C07287=1050.995,70.390,419.955,170.839,33.457,156.282
C07288=1051.001,70.640,419.937,170.841,33.459,156.283
C07289=1051.007,70.890,419.919,170.843,33.461,156.283
C07290=1051.013,71.138,419.901,170.844,33.463,156.283
C07291=1051.019,71.388,419.883,170.846,33.465,156.284
C07292=1051.025,71.638,419.865,170.847,33.467,156.284
C07293=1051.031,71.887,419.846,170.849,33.469,156.284
C07294=1051.037,72.136,419.828,170.851,33.471,156.285
C07295=1051.044,72.385,419.810,170.852,33.473,156.285
C07296=1051.050,72.635,419.792,170.854,33.475,156.285
C07297=1051.056,72.884,419.775,170.856,33.478,156.286
C07298=1051.062,73.133,419.756,170.857,33.479,156.286
C07299=1051.068,73.382,419.738,170.859,33.481,156.286
C07300=1051.075,73.632,419.720,170.861,33.483,156.287
C07301=1051.080,73.881,419.702,170.863,33.485,156.287
C07302=1051.086,74.130,419.684,170.865,33.487,156.287
C07303=1051.093,74.379,419.665,170.866,33.490,156.288
C07304=1051.099,74.629,419.648,170.868,33.492,156.288
C07305=1051.105,74.878,419.629,170.870,33.494,156.288
C07306=1051.111,75.127,419.611,170.871,33.496,156.289
C07307=1051.117,75.376,419.593,170.873,33.498,156.289
C07308=1051.124,75.626,419.575,170.874,33.500,156.289
C07309=1051.130,75.874,419.557,170.876,33.502,156.290
C07310=1051.136,76.124,419.539,170.878,33.504,156.290
C07311=1051.142,76.373,419.520,170.879,33.506,156.291
C07312=1051.148,76.623,419.503,170.881,33.508,156.291
C07313=1051.154,76.871,419.484,170.883,33.510,156.291
C07314=1051.160,77.121,419.466,170.884,33.512,156.291
C07315=1051.167,77.407,419.445,170.886,33.515,156.292
C07316=1051.175,77.693,419.424,170.888,33.517,156.292
C07317=1051.182,77.978,419.403,170.890,33.519,156.293
C07318=1051.189,78.264,419.382,170.892,33.522,156.293
C07319=1051.195,78.513,419.364,170.893,33.524,156.293
C07320=1051.201,78.762,419.346,170.895,33.526,156.294
C07321=1051.207,79.011,419.327,170.897,33.528,156.294
C07322=1051.213,79.261,419.309,170.898,33.530,156.294
C07323=1051.219,79.510,419.290,170.900,33.532,156.295
C07324=1051.225,79.759,419.271,170.901,33.534,156.295
C07325=1051.231,80.009,419.254,170.903,33.536,156.295
C07326=1051.237,80.257,419.235,170.905,33.538,156.296
C07327=1051.244,80.506,419.217,170.906,33.541,156.296
C07328=1051.250,80.756,419.199,170.908,33.543,156.297
C07329=1051.255,81.006,419.179,170.909,33.545,156.297
C07330=1051.262,81.255,419.161,170.911,33.547,156.297
C07331=1051.267,81.504,419.143,170.913,33.549,156.298
C07332=1051.274,81.753,419.125,170.914,33.551,156.298
C07333=1051.280,82.002,419.106,170.916,33.553,156.298
C07334=1051.286,82.252,419.087,170.918,33.555,156.299
C07335=1051.292,82.501,419.069,170.919,33.558,156.299
C07336=1051.298,82.750,419.050,170.921,33.560,156.299
C07337=1051.304,82.999,419.032,170.922,33.562,156.300
C07338=1051.310,83.249,419.014,170.924,33.564,156.300
C07339=1051.316,83.498,418.995,170.926,33.566,156.300
C07340=1051.322,83.747,418.976,170.927,33.568,156.301
C07341=1051.329,83.996,418.957,170.929,33.570,156.301
C07342=1051.335,84.246,418.939,170.931,33.572,156.301
C07343=1051.340,84.495,418.920,170.933,33.574,156.302
C07344=1051.347,84.744,418.902,170.935,33.576,156.302
C07345=1051.353,84.993,418.883,170.936,33.579,156.302
C07346=1051.359,85.242,418.865,170.938,33.580,156.303
C07347=1051.365,85.492,418.847,170.940,33.582,156.303
C07348=1051.371,85.741,418.827,170.941,33.584,156.303
C07349=1051.378,85.990,418.809,170.943,33.586,156.304
C07350=1051.384,86.239,418.790,170.945,33.589,156.304
C07351=1051.390,86.489,418.771,170.946,33.591,156.304
C07352=1051.396,86.738,418.752,170.948,33.593,156.305
C07353=1051.402,86.987,418.735,170.949,33.595,156.305
C07354=1051.408,87.236,418.716,170.951,33.597,156.305
C07355=1051.415,87.485,418.697,170.953,33.599,156.306
C07356=1051.420,87.735,418.678,170.954,33.601,156.306
C07357=1051.427,87.984,418.659,170.956,33.603,156.307
C07358=1051.433,88.233,418.641,170.958,33.605,156.307
C07359=1051.439,88.482,418.622,170.959,33.607,156.307
C07360=1051.445,88.732,418.603,170.961,33.609,156.307
C07361=1051.452,88.981,418.584,170.963,33.612,156.308
C07362=1051.458,89.230,418.566,170.964,33.614,156.308
C07363=1051.464,89.480,418.548,170.966,33.616,156.309
C07364=1051.470,89.729,418.528,170.968,33.618,156.309
C07365=1051.476,89.978,418.510,170.969,33.620,156.309
C07366=1051.483,90.227,418.491,170.971,33.622,156.310
C07367=1051.489,90.476,418.472,170.972,33.624,156.310
C07368=1051.495,90.726,418.453,170.974,33.626,156.310
C07369=1051.501,90.975,418.435,170.976,33.628,156.311
C07370=1051.507,91.224,418.415,170.977,33.631,156.311
C07371=1051.513,91.473,418.397,170.979,33.633,156.311
C07372=1051.519,91.723,418.377,170.981,33.634,156.312
C07373=1051.525,91.972,418.359,170.982,33.636,156.312
C07374=1051.531,92.221,418.340,170.984,33.639,156.312
C07375=1051.537,92.469,418.321,170.985,33.641,156.313
C07376=1051.543,92.719,418.301,170.988,33.643,156.313
C07377=1051.549,92.968,418.283,170.990,33.645,156.314
C07378=1051.555,93.217,418.263,170.991,33.647,156.314
C07379=1051.562,93.504,418.242,170.993,33.650,156.314
C07380=1051.569,93.789,418.220,170.995,33.652,156.315
C07381=1051.576,94.075,418.198,170.997,33.655,156.315
C07382=1051.583,94.360,418.176,170.999,33.657,156.315
C07383=1051.589,94.609,418.158,171.000,33.659,156.316
C07384=1051.595,94.858,418.138,171.002,33.662,156.316
C07385=1051.602,95.107,418.119,171.004,33.664,156.317
C07386=1051.608,95.356,418.100,171.005,33.666,156.317
C07387=1051.613,95.606,418.080,171.007,33.667,156.317
C07388=1051.620,95.855,418.062,171.009,33.670,156.318
C07389=1051.625,96.104,418.043,171.010,33.672,156.318
C07390=1051.632,96.353,418.024,171.012,33.674,156.318
C07391=1051.638,96.602,418.004,171.014,33.676,156.319
C07392=1051.644,96.851,417.985,171.015,33.678,156.319
C07393=1051.650,97.101,417.966,171.017,33.680,156.319
C07394=1051.656,97.350,417.947,171.019,33.682,156.320
C07395=1051.662,97.599,417.928,171.020,33.684,156.320
C07396=1051.669,97.848,417.909,171.022,33.687,156.320
C07397=1051.674,98.097,417.890,171.024,33.689,156.321
C07398=1051.680,98.347,417.870,171.025,33.691,156.321
C07399=1051.687,98.597,417.851,171.027,33.693,156.321
C07400=1051.693,98.845,417.831,171.028,33.695,156.322
C07401=1051.700,99.094,417.813,171.030,33.697,156.322
C07402=1051.705,99.344,417.793,171.032,33.699,156.323
C07403=1051.712,99.592,417.774,171.033,33.701,156.323
C07404=1051.718,99.842,417.755,171.036,33.704,156.323
C07405=1051.724,100.091,417.736,171.038,33.706,156.324
C07406=1051.730,100.340,417.717,171.039,33.708,156.324
C07407=1051.736,100.589,417.697,171.041,33.710,156.324
C07408=1051.742,100.838,417.678,171.043,33.712,156.325
C07409=1051.748,101.088,417.659,171.044,33.714,156.325
C07410=1051.754,101.337,417.639,171.046,33.716,156.325
C07411=1051.760,101.587,417.620,171.048,33.719,156.326
C07412=1051.767,101.835,417.600,171.049,33.721,156.326
C07413=1051.773,102.085,417.581,171.051,33.723,156.326
C07414=1051.778,102.334,417.562,171.053,33.725,156.327
C07415=1051.784,102.583,417.542,171.054,33.727,156.327
C07416=1051.790,102.832,417.522,171.056,33.729,156.328
C07417=1051.797,103.081,417.503,171.058,33.732,156.328
C07418=1051.802,103.330,417.484,171.059,33.733,156.328
C07419=1051.808,103.579,417.464,171.061,33.735,156.329
C07420=1051.814,103.829,417.445,171.062,33.738,156.329
C07421=1051.821,104.078,417.424,171.064,33.740,156.329
C07422=1051.826,104.327,417.405,171.066,33.742,156.330
C07423=1051.833,104.576,417.386,171.067,33.744,156.330
C07424=1051.839,104.825,417.367,171.069,33.746,156.330
C07425=1051.845,105.074,417.347,171.071,33.748,156.331
C07426=1051.850,105.324,417.327,171.072,33.751,156.331
C07427=1051.856,105.572,417.307,171.074,33.753,156.332
C07428=1051.863,105.822,417.289,171.076,33.755,156.332
C07429=1051.869,106.071,417.268,171.078,33.757,156.332
C07430=1051.875,106.321,417.249,171.080,33.759,156.333
C07431=1051.881,106.569,417.229,171.082,33.761,156.333
C07432=1051.887,106.819,417.210,171.083,33.764,156.333
C07433=1051.893,107.068,417.190,171.085,33.766,156.334
C07434=1051.899,107.317,417.171,171.087,33.768,156.334
C07435=1051.906,107.566,417.151,171.088,33.770,156.335
C07436=1051.912,107.815,417.131,171.090,33.772,156.335
C07437=1051.918,108.064,417.112,171.092,33.774,156.335
C07438=1051.924,108.313,417.092,171.093,33.777,156.336
C07439=1051.929,108.563,417.073,171.095,33.779,156.336
C07440=1051.936,108.812,417.052,171.097,33.781,156.336
C07441=1051.943,109.061,417.033,171.098,33.783,156.337
C07442=1051.948,109.310,417.014,171.100,33.785,156.337
C07443=1051.955,109.596,416.991,171.102,33.788,156.337
C07444=1051.963,109.881,416.968,171.104,33.790,156.338
C07445=1051.970,110.166,416.946,171.106,33.792,156.338
C07446=1051.976,110.452,416.923,171.108,33.795,156.339
C07447=1051.982,110.701,416.903,171.110,33.797,156.339
C07448=1051.988,110.951,416.883,171.111,33.799,156.339
C07449=1051.994,111.200,416.863,171.113,33.801,156.340
C07450=1052.000,111.449,416.843,171.115,33.803,156.340
C07451=1052.006,111.698,416.824,171.117,33.806,156.341
C07452=1052.012,111.947,416.804,171.119,33.808,156.341
C07453=1052.019,112.197,416.784,171.121,33.810,156.341
C07454=1052.025,112.445,416.764,171.122,33.812,156.342
C07455=1052.030,112.695,416.745,171.124,33.814,156.342
C07456=1052.036,112.944,416.725,171.126,33.816,156.342
C07457=1052.043,113.193,416.704,171.127,33.819,156.343
C07458=1052.049,113.442,416.684,171.129,33.821,156.343
C07459=1052.055,113.691,416.665,171.131,33.823,156.343
C07460=1052.061,113.940,416.645,171.132,33.825,156.344
C07461=1052.067,114.190,416.625,171.134,33.827,156.344
C07462=1052.073,114.439,416.605,171.136,33.830,156.345
C07463=1052.079,114.688,416.584,171.137,33.831,156.345
C07464=1052.085,114.936,416.564,171.139,33.834,156.345
C07465=1052.091,115.186,416.544,171.141,33.836,156.346
C07466=1052.097,115.435,416.525,171.142,33.838,156.346
C07467=1052.102,115.685,416.504,171.144,33.840,156.346
C07468=1052.108,115.933,416.484,171.146,33.843,156.347
C07469=1052.115,116.183,416.464,171.147,33.845,156.347
C07470=1052.121,116.432,416.444,171.149,33.847,156.348
C07471=1052.126,116.681,416.423,171.152,33.849,156.348
C07472=1052.132,116.930,416.403,171.154,33.852,156.348
C07473=1052.139,117.179,416.383,171.155,33.854,156.349
C07474=1052.144,117.428,416.363,171.157,33.856,156.349
C07475=1052.150,117.677,416.343,171.159,33.858,156.349
C07476=1052.156,117.926,416.323,171.160,33.860,156.350
C07477=1052.162,118.175,416.302,171.162,33.863,156.350
C07478=1052.168,118.424,416.282,171.164,33.865,156.351
C07479=1052.174,118.673,416.262,171.165,33.867,156.351
C07480=1052.180,118.923,416.241,171.167,33.869,156.351
C07481=1052.186,119.172,416.221,171.169,33.872,156.352
C07482=1052.191,119.421,416.201,171.170,33.874,156.352
C07483=1052.197,119.670,416.181,171.172,33.876,156.352
C07484=1052.204,119.919,416.161,171.174,33.878,156.353
C07485=1052.210,120.168,416.141,171.176,33.880,156.353
C07486=1052.215,120.417,416.120,171.177,33.883,156.354
C07487=1052.222,120.667,416.100,171.179,33.885,156.354
C07488=1052.228,120.915,416.080,171.181,33.887,156.354
C07489=1052.233,121.165,416.059,171.182,33.889,156.355
C07490=1052.240,121.414,416.039,171.185,33.892,156.355
C07491=1052.246,121.663,416.019,171.187,33.894,156.356
C07492=1052.252,121.912,415.997,171.188,33.896,156.356
C07493=1052.258,122.161,415.977,171.190,33.898,156.356
C07494=1052.264,122.410,415.957,171.192,33.900,156.357
C07495=1052.270,122.659,415.937,171.194,33.903,156.357
C07496=1052.276,122.908,415.917,171.195,33.905,156.357
C07497=1052.282,123.157,415.897,171.197,33.907,156.358
C07498=1052.288,123.407,415.876,171.199,33.909,156.358
C07499=1052.294,123.656,415.856,171.200,33.911,156.358
C07500=1052.300,123.905,415.835,171.202,33.914,156.359
C07501=1052.306,124.153,415.815,171.204,33.916,156.359
C07502=1052.312,124.403,415.794,171.206,33.918,156.360
C07503=1052.318,124.652,415.774,171.207,33.920,156.360
C07504=1052.324,124.901,415.754,171.209,33.922,156.360
C07505=1052.330,125.150,415.732,171.211,33.925,156.361
C07506=1052.336,125.399,415.712,171.213,33.926,156.361
C07507=1052.343,125.684,415.689,171.215,33.929,156.362
C07508=1052.350,125.970,415.666,171.218,33.932,156.362
C07509=1052.357,126.256,415.642,171.220,33.934,156.362
C07510=1052.364,126.541,415.618,171.222,33.937,156.363
C07511=1052.370,126.790,415.598,171.223,33.939,156.363
C07512=1052.377,127.039,415.577,171.225,33.941,156.364
C07513=1052.382,127.288,415.557,171.227,33.943,156.364
C07514=1052.389,127.537,415.537,171.229,33.945,156.364
C07515=1052.394,127.786,415.515,171.230,33.948,156.365
C07516=1052.401,128.036,415.495,171.232,33.950,156.365
C07517=1052.407,128.284,415.475,171.234,33.952,156.366
C07518=1052.413,128.534,415.454,171.236,33.954,156.366
C07519=1052.419,128.782,415.433,171.237,33.956,156.366
C07520=1052.426,129.032,415.413,171.239,33.958,156.367
C07521=1052.431,129.281,415.392,171.241,33.960,156.367
C07522=1052.438,129.530,415.371,171.243,33.963,156.367
C07523=1052.444,129.779,415.352,171.244,33.965,156.368
C07524=1052.450,130.028,415.330,171.246,33.967,156.368
C07525=1052.456,130.277,415.310,171.249,33.969,156.369
C07526=1052.462,130.527,415.289,171.251,33.971,156.369
C07527=1052.468,130.775,415.268,171.252,33.973,156.369
C07528=1052.475,131.024,415.248,171.254,33.976,156.370
C07529=1052.481,131.273,415.226,171.256,33.978,156.370
C07530=1052.487,131.522,415.206,171.258,33.980,156.370
C07531=1052.493,131.772,415.185,171.259,33.982,156.371
C07532=1052.499,132.020,415.165,171.261,33.985,156.371
C07533=1052.505,132.270,415.144,171.263,33.987,156.371
C07534=1052.511,132.519,415.123,171.265,33.989,156.372
C07535=1052.517,132.768,415.102,171.266,33.991,156.372
C07536=1052.523,133.017,415.081,171.268,33.994,156.373
C07537=1052.529,133.266,415.060,171.270,33.996,156.373
C07538=1052.535,133.515,415.039,171.272,33.998,156.373
C07539=1052.541,133.764,415.018,171.273,34.000,156.374
C07540=1052.546,134.013,414.997,171.275,34.003,156.374
C07541=1052.553,134.262,414.976,171.278,34.005,156.375
C07542=1052.559,134.511,414.956,171.280,34.007,156.375
C07543=1052.565,134.760,414.934,171.282,34.009,156.375
C07544=1052.571,135.009,414.914,171.283,34.012,156.376
C07545=1052.577,135.258,414.892,171.285,34.014,156.376
C07546=1052.582,135.507,414.871,171.287,34.016,156.377
C07547=1052.589,135.756,414.851,171.289,34.018,156.377
C07548=1052.595,136.005,414.829,171.290,34.021,156.377
C07549=1052.600,136.255,414.809,171.292,34.022,156.378
C07550=1052.607,136.503,414.788,171.294,34.025,156.378
C07551=1052.613,136.752,414.766,171.296,34.027,156.378
C07552=1052.619,137.002,414.745,171.298,34.030,156.379
C07553=1052.625,137.250,414.725,171.299,34.031,156.379
C07554=1052.631,137.499,414.703,171.301,34.034,156.380
C07555=1052.637,137.749,414.682,171.303,34.036,156.380
C07556=1052.643,137.998,414.661,171.306,34.038,156.380
C07557=1052.650,138.246,414.640,171.307,34.041,156.381
C07558=1052.655,138.496,414.619,171.309,34.043,156.381
C07559=1052.661,138.745,414.598,171.311,34.045,156.382
C07560=1052.667,138.994,414.576,171.313,34.047,156.382
C07561=1052.673,139.242,414.555,171.315,34.050,156.382
C07562=1052.679,139.492,414.534,171.316,34.052,156.383
C07563=1052.685,139.741,414.513,171.318,34.054,156.383
C07564=1052.691,139.990,414.492,171.320,34.056,156.384
C07565=1052.697,140.239,414.470,171.322,34.059,156.384
C07566=1052.702,140.488,414.449,171.324,34.061,156.384
C07567=1052.709,140.737,414.428,171.325,34.063,156.385
C07568=1052.715,140.986,414.407,171.327,34.066,156.385
C07569=1052.721,141.235,414.385,171.329,34.068,156.386
C07570=1052.727,141.484,414.364,171.332,34.070,156.386
C07571=1052.733,141.770,414.340,171.334,34.073,156.386
C07572=1052.741,142.054,414.315,171.336,34.075,156.387
C07573=1052.747,142.339,414.290,171.338,34.078,156.387
C07574=1052.754,142.625,414.266,171.340,34.081,156.388
C07575=1052.760,142.874,414.244,171.342,34.083,156.388
C07576=1052.767,143.123,414.223,171.344,34.086,156.389
C07577=1052.772,143.372,414.202,171.345,34.088,156.389
C07578=1052.778,143.621,414.180,171.347,34.090,156.389
C07579=1052.785,143.870,414.159,171.349,34.092,156.390
C07580=1052.790,144.119,414.137,171.351,34.095,156.390
C07581=1052.796,144.368,414.116,171.353,34.097,156.391
C07582=1052.802,144.617,414.094,171.355,34.099,156.391
C07583=1052.808,144.866,414.074,171.357,34.102,156.391
C07584=1052.814,145.115,414.052,171.359,34.103,156.392
C07585=1052.820,145.365,414.030,171.361,34.106,156.392
C07586=1052.826,145.614,414.009,171.363,34.108,156.393
C07587=1052.832,145.862,413.987,171.365,34.111,156.393
C07588=1052.838,146.111,413.966,171.367,34.113,156.393
C07589=1052.844,146.361,413.944,171.368,34.115,156.394
C07590=1052.850,146.609,413.923,171.370,34.117,156.394
C07591=1052.856,146.858,413.901,171.372,34.119,156.395
C07592=1052.862,147.108,413.880,171.374,34.122,156.395
C07593=1052.868,147.357,413.858,171.376,34.124,156.395
C07594=1052.874,147.605,413.836,171.378,34.126,156.396
C07595=1052.880,147.854,413.814,171.379,34.129,156.396
C07596=1052.886,148.103,413.793,171.381,34.131,156.397
C07597=1052.892,148.352,413.771,171.384,34.133,156.397
C07598=1052.898,148.601,413.750,171.386,34.136,156.397
C07599=1052.904,148.850,413.728,171.388,34.138,156.398
C07600=1052.910,149.099,413.707,171.390,34.140,156.398
C07601=1052.917,149.348,413.685,171.391,34.143,156.399
C07602=1052.922,149.597,413.664,171.393,34.145,156.399
C07603=1052.928,149.846,413.641,171.395,34.147,156.399
C07604=1052.934,150.095,413.619,171.397,34.150,156.400
C07605=1052.940,150.344,413.597,171.399,34.152,156.400
C07606=1052.946,150.593,413.576,171.401,34.154,156.401
C07607=1052.952,150.842,413.555,171.403,34.157,156.401
C07608=1052.958,151.090,413.532,171.404,34.159,156.401
C07609=1052.964,151.340,413.510,171.407,34.161,156.402
C07610=1052.970,151.589,413.488,171.409,34.164,156.402
C07611=1052.975,151.838,413.467,171.411,34.166,156.403
C07612=1052.982,152.086,413.445,171.413,34.168,156.403
C07613=1052.988,152.336,413.423,171.415,34.171,156.404
C07614=1052.994,152.585,413.401,171.417,34.173,156.404
C07615=1053.000,152.834,413.379,171.418,34.175,156.404
C07616=1053.006,153.082,413.357,171.420,34.178,156.405
C07617=1053.012,153.331,413.336,171.422,34.180,156.405
C07618=1053.018,153.581,413.314,171.424,34.182,156.406
C07619=1053.023,153.830,413.292,171.426,34.185,156.406
C07620=1053.030,154.079,413.269,171.428,34.187,156.406
C07621=1053.036,154.328,413.248,171.431,34.189,156.407
C07622=1053.042,154.576,413.226,171.433,34.192,156.407
C07623=1053.047,154.825,413.204,171.434,34.194,156.408
C07624=1053.053,155.074,413.182,171.436,34.196,156.408
C07625=1053.060,155.323,413.160,171.438,34.199,156.409
C07626=1053.065,155.573,413.137,171.440,34.201,156.409
C07627=1053.071,155.822,413.116,171.442,34.203,156.409
C07628=1053.077,156.070,413.094,171.444,34.206,156.410
C07629=1053.083,156.319,413.071,171.446,34.208,156.410
C07630=1053.089,156.568,413.049,171.448,34.211,156.411
C07631=1053.095,156.817,413.027,171.450,34.213,156.411
C07632=1053.101,157.066,413.005,171.451,34.215,156.411
C07633=1053.107,157.315,412.983,171.454,34.218,156.412
C07634=1053.113,157.564,412.961,171.456,34.220,156.412
C07635=1053.120,157.849,412.936,171.458,34.223,156.413
C07636=1053.127,158.134,412.911,171.461,34.225,156.413
C07637=1053.134,158.418,412.885,171.463,34.228,156.414
C07638=1053.141,158.704,412.860,171.465,34.231,156.414
C07639=1053.146,158.952,412.837,171.467,34.233,156.415
C07640=1053.152,159.201,412.815,171.469,34.236,156.415
C07641=1053.158,159.450,412.792,171.471,34.238,156.415
C07642=1053.164,159.700,412.771,171.473,34.241,156.416
C07643=1053.171,159.948,412.748,171.475,34.243,156.416
C07644=1053.176,160.198,412.726,171.477,34.245,156.417
C07645=1053.183,160.446,412.704,171.479,34.248,156.417
C07646=1053.189,160.695,412.682,171.481,34.250,156.417
C07647=1053.194,160.944,412.659,171.483,34.252,156.418
C07648=1053.200,161.193,412.636,171.485,34.255,156.418
C07649=1053.206,161.443,412.614,171.487,34.257,156.419
C07650=1053.212,161.691,412.592,171.489,34.260,156.419
C07651=1053.217,161.940,412.569,171.491,34.262,156.420
C07652=1053.223,162.189,412.547,171.493,34.265,156.420
C07653=1053.228,162.438,412.524,171.495,34.267,156.421
C07654=1053.235,162.687,412.502,171.498,34.270,156.421
C07655=1053.241,162.935,412.479,171.499,34.272,156.422
C07656=1053.246,163.185,412.456,171.501,34.275,156.422
C07657=1053.252,163.434,412.434,171.503,34.277,156.422
C07658=1053.258,163.682,412.411,171.505,34.280,156.423
C07659=1053.264,163.931,412.388,171.507,34.282,156.423
C07660=1053.269,164.181,412.366,171.509,34.285,156.424
C07661=1053.274,164.429,412.343,171.511,34.287,156.424
C07662=1053.281,164.678,412.321,171.513,34.289,156.425
C07663=1053.287,164.927,412.298,171.515,34.292,156.425
C07664=1053.292,165.175,412.275,171.517,34.294,156.425
C07665=1053.298,165.425,412.253,171.520,34.297,156.426
C07666=1053.304,165.674,412.231,171.522,34.299,156.426
C07667=1053.310,165.922,412.208,171.524,34.302,156.427
C07668=1053.316,166.171,412.185,171.525,34.304,156.427
C07669=1053.321,166.420,412.162,171.527,34.307,156.428
C07670=1053.327,166.669,412.139,171.529,34.309,156.428
C07671=1053.334,166.918,412.116,171.531,34.312,156.429
C07672=1053.339,167.167,412.094,171.533,34.315,156.429
C07673=1053.345,167.416,412.071,171.535,34.317,156.430
C07674=1053.351,167.665,412.048,171.538,34.320,156.430
C07675=1053.357,167.914,412.026,171.540,34.322,156.430
C07676=1053.363,168.162,412.003,171.542,34.324,156.431
C07677=1053.368,168.411,411.980,171.544,34.327,156.431
C07678=1053.374,168.660,411.957,171.546,34.329,156.432
C07679=1053.380,168.909,411.934,171.548,34.332,156.432
C07680=1053.386,169.158,411.911,171.550,34.334,156.433
C07681=1053.392,169.407,411.889,171.552,34.337,156.433
C07682=1053.398,169.656,411.866,171.554,34.339,156.433
C07683=1053.404,169.904,411.843,171.556,34.342,156.434
C07684=1053.409,170.153,411.820,171.559,34.344,156.434
C07685=1053.415,170.402,411.797,171.561,34.347,156.435
C07686=1053.422,170.651,411.775,171.563,34.349,156.435
C07687=1053.428,170.900,411.751,171.565,34.352,156.436
C07688=1053.434,171.149,411.729,171.567,34.354,156.436
C07689=1053.439,171.398,411.706,171.569,34.357,156.437
C07690=1053.445,171.647,411.683,171.571,34.359,156.437
C07691=1053.451,171.896,411.660,171.573,34.362,156.438
C07692=1053.457,172.145,411.637,171.575,34.364,156.438
C07693=1053.463,172.393,411.614,171.577,34.366,156.438
C07694=1053.469,172.642,411.591,171.580,34.369,156.439
C07695=1053.474,172.891,411.568,171.582,34.371,156.439
C07696=1053.481,173.141,411.545,171.584,34.374,156.440
C07697=1053.487,173.389,411.522,171.586,34.376,156.440
C07698=1053.493,173.638,411.499,171.588,34.379,156.441
C07699=1053.499,173.923,411.473,171.590,34.382,156.441
C07700=1053.507,174.206,411.446,171.592,34.384,156.442
C07701=1053.513,174.492,411.420,171.595,34.388,156.442
C07702=1053.520,174.776,411.394,171.597,34.390,156.443
C07703=1053.526,175.025,411.371,171.600,34.393,156.443
C07704=1053.532,175.273,411.348,171.602,34.395,156.444
C07705=1053.538,175.522,411.325,171.604,34.398,156.444
C07706=1053.544,175.772,411.301,171.606,34.400,156.444
C07707=1053.550,176.021,411.278,171.608,34.403,156.445
C07708=1053.557,176.269,411.255,171.610,34.405,156.445
C07709=1053.562,176.518,411.232,171.612,34.408,156.446
C07710=1053.568,176.767,411.209,171.614,34.410,156.446
C07711=1053.574,177.016,411.186,171.616,34.413,156.447
C07712=1053.580,177.264,411.162,171.620,34.415,156.447
C07713=1053.586,177.513,411.139,171.622,34.418,156.448
C07714=1053.592,177.762,411.117,171.624,34.420,156.448
C07715=1053.599,178.011,411.093,171.626,34.423,156.449
C07716=1053.605,178.260,411.070,171.628,34.425,156.449
C07717=1053.611,178.509,411.047,171.630,34.427,156.449
C07718=1053.617,178.757,411.024,171.632,34.430,156.450
C07719=1053.623,179.007,411.000,171.634,34.432,156.450
C07720=1053.629,179.255,410.977,171.636,34.435,156.451
C07721=1053.635,179.504,410.954,171.639,34.437,156.451
C07722=1053.641,179.753,410.931,171.641,34.440,156.452
C07723=1053.647,180.002,410.907,171.643,34.442,156.452
C07724=1053.653,180.251,410.884,171.645,34.445,156.453
C07725=1053.659,180.499,410.861,171.647,34.447,156.453
C07726=1053.665,180.748,410.837,171.650,34.450,156.453
C07727=1053.672,180.997,410.814,171.652,34.452,156.454
C07728=1053.678,181.246,410.791,171.654,34.455,156.454
C07729=1053.684,181.495,410.767,171.656,34.457,156.455
C07730=1053.690,181.744,410.744,171.659,34.460,156.455
C07731=1053.696,181.992,410.721,171.661,34.462,156.456
C07732=1053.702,182.242,410.697,171.663,34.465,156.456
C07733=1053.708,182.490,410.674,171.665,34.468,156.457
C07734=1053.714,182.739,410.651,171.667,34.470,156.457
C07735=1053.721,182.988,410.627,171.669,34.473,156.458
C07736=1053.726,183.237,410.604,171.672,34.475,156.458
C07737=1053.733,183.486,410.580,171.674,34.478,156.458
C07738=1053.739,183.735,410.557,171.677,34.480,156.459
C07739=1053.745,183.983,410.533,171.679,34.483,156.459
C07740=1053.751,184.232,410.510,171.681,34.485,156.460
C07741=1053.757,184.481,410.486,171.683,34.488,156.460
C07742=1053.762,184.729,410.462,171.685,34.490,156.461
C07743=1053.769,184.979,410.439,171.687,34.493,156.461
C07744=1053.775,185.227,410.415,171.689,34.496,156.462
C07745=1053.780,185.476,410.391,171.691,34.498,156.462
C07746=1053.786,185.725,410.368,171.695,34.501,156.463
C07747=1053.792,185.974,410.343,171.697,34.504,156.463
C07748=1053.798,186.222,410.320,171.699,34.506,156.464
C07749=1053.803,186.471,410.295,171.701,34.509,156.464
C07750=1053.809,186.720,410.272,171.703,34.512,156.465
C07751=1053.815,186.969,410.248,171.705,34.514,156.465
C07752=1053.821,187.217,410.224,171.707,34.517,156.466
C07753=1053.827,187.466,410.200,171.709,34.519,156.466
C07754=1053.832,187.715,410.177,171.712,34.523,156.467
C07755=1053.838,187.964,410.153,171.715,34.525,156.467
C07756=1053.844,188.213,410.128,171.717,34.528,156.468
C07757=1053.850,188.461,410.105,171.719,34.531,156.468
C07758=1053.856,188.710,410.080,171.721,34.533,156.469
C07759=1053.862,188.959,410.057,171.723,34.536,156.469
C07760=1053.867,189.208,410.033,171.725,34.538,156.470
C07761=1053.873,189.456,410.009,171.728,34.541,156.470
C07762=1053.879,189.706,409.984,171.730,34.544,156.471
C07763=1053.886,189.990,409.957,171.733,34.547,156.471
C07764=1053.892,190.273,409.930,171.735,34.550,156.472
C07765=1053.900,190.558,409.902,171.738,34.553,156.472
C07766=1053.906,190.842,409.875,171.740,34.556,156.473
C07767=1053.912,191.090,409.851,171.742,34.559,156.473
C07768=1053.918,191.339,409.826,171.746,34.561,156.474
C07769=1053.924,191.587,409.803,171.748,34.564,156.474
C07770=1053.930,191.837,409.779,171.750,34.567,156.475
C07771=1053.936,192.086,409.755,171.752,34.569,156.475
C07772=1053.942,192.335,409.731,171.754,34.573,156.476
C07773=1053.948,192.583,409.707,171.756,34.575,156.476
C07774=1053.954,192.833,409.682,171.759,34.578,156.477
C07775=1053.960,193.081,409.659,171.761,34.581,156.477
C07776=1053.966,193.330,409.634,171.764,34.583,156.478
C07777=1053.972,193.578,409.610,171.766,34.586,156.478
C07778=1053.978,193.827,409.585,171.768,34.589,156.479
C07779=1053.984,194.075,409.561,171.770,34.591,156.479
C07780=1053.990,194.325,409.537,171.773,34.594,156.480
C07781=1053.996,194.573,409.513,171.775,34.597,156.480
C07782=1054.002,194.822,409.488,171.777,34.599,156.481
C07783=1054.007,195.071,409.464,171.780,34.602,156.481
C07784=1054.014,195.320,409.440,171.782,34.605,156.482
C07785=1054.019,195.568,409.416,171.785,34.608,156.482
C07786=1054.026,195.817,409.392,171.787,34.610,156.483
C07787=1054.031,196.066,409.368,171.789,34.613,156.483
C07788=1054.038,196.314,409.343,171.791,34.616,156.484
C07789=1054.043,196.563,409.319,171.793,34.618,156.484
C07790=1054.050,196.812,409.295,171.797,34.621,156.485
C07791=1054.056,197.061,409.270,171.799,34.624,156.485
C07792=1054.062,197.309,409.246,171.801,34.627,156.486
C07793=1054.068,197.559,409.222,171.803,34.629,156.486
C07794=1054.073,197.807,409.197,171.806,34.632,156.487
C07795=1054.080,198.056,409.173,171.808,34.635,156.487
C07796=1054.085,198.304,409.148,171.810,34.637,156.488
C07797=1054.092,198.553,409.124,171.813,34.640,156.488
C07798=1054.098,198.802,409.099,171.815,34.643,156.489
C07799=1054.104,199.050,409.075,171.818,34.646,156.489
C07800=1054.110,199.299,409.051,171.820,34.649,156.490
C07801=1054.116,199.549,409.026,171.822,34.651,156.490
C07802=1054.122,199.796,409.002,171.824,34.654,156.491
C07803=1054.128,200.046,408.977,171.827,34.657,156.491
C07804=1054.135,200.295,408.953,171.830,34.659,156.492
C07805=1054.140,200.543,408.928,171.832,34.662,156.492
C07806=1054.147,200.792,408.904,171.835,34.665,156.493
C07807=1054.153,201.041,408.880,171.837,34.667,156.493
C07808=1054.159,201.289,408.855,171.839,34.670,156.494
C07809=1054.165,201.538,408.831,171.841,34.673,156.494
C07810=1054.171,201.786,408.805,171.845,34.676,156.495
C07811=1054.177,202.035,408.781,171.847,34.678,156.495
C07812=1054.183,202.284,408.756,171.849,34.682,156.496
C07813=1054.189,202.533,408.732,171.851,34.684,156.496
C07814=1054.195,202.781,408.707,171.854,34.687,156.497
C07815=1054.201,203.030,408.682,171.856,34.690,156.498
C07816=1054.206,203.279,408.658,171.858,34.693,156.498
C07817=1054.213,203.527,408.632,171.861,34.696,156.499
C07818=1054.218,203.777,408.608,171.864,34.698,156.499
C07819=1054.224,204.024,408.583,171.866,34.701,156.500
C07820=1054.230,204.273,408.557,171.868,34.705,156.500
C07821=1054.236,204.522,408.533,171.870,34.707,156.501
C07822=1054.242,204.771,408.507,171.873,34.710,156.501
C07823=1054.248,205.019,408.484,171.876,34.713,156.502
C07824=1054.255,205.268,408.458,171.878,34.716,156.502
C07825=1054.260,205.517,408.434,171.881,34.719,156.503
C07826=1054.266,205.765,408.409,171.883,34.721,156.503
C07827=1054.291,206.816,408.303,172.092,34.813,156.518
C07828=1054.298,207.059,408.278,172.094,34.817,156.519
C07829=1054.304,207.301,408.252,172.096,34.821,156.520
C07830=1054.311,207.543,408.228,172.098,34.824,156.520
C07831=1054.316,207.785,408.203,172.100,34.828,156.521
C07832=1054.323,208.027,408.177,172.101,34.832,156.522
C07833=1054.329,208.269,408.152,172.104,34.835,156.523
C07834=1054.335,208.511,408.127,172.106,34.839,156.523
C07835=1054.341,208.753,408.102,172.107,34.842,156.524
C07836=1054.347,209.001,408.076,172.109,34.846,156.525
C07837=1054.353,209.251,408.049,172.112,34.850,156.525
C07838=1054.360,209.499,408.023,172.114,34.853,156.526
C07839=1054.366,209.748,407.998,172.115,34.857,156.527
C07840=1054.373,209.996,407.972,172.117,34.861,156.528
C07841=1054.379,210.245,407.945,172.120,34.864,156.528
C07842=1054.385,210.493,407.919,172.122,34.868,156.529
C07843=1054.392,210.741,407.893,172.123,34.872,156.530
C07844=1054.397,210.990,407.867,172.125,34.876,156.530
C07845=1054.404,211.239,407.841,172.128,34.879,156.531
C07846=1054.410,211.488,407.814,172.130,34.883,156.532
C07847=1054.416,211.736,407.789,172.131,34.886,156.533
C07848=1054.423,211.984,407.763,172.133,34.890,156.533
C07849=1054.429,212.233,407.736,172.136,34.894,156.534
C07850=1054.436,212.481,407.710,172.138,34.897,156.535
C07851=1054.441,212.730,407.684,172.139,34.901,156.535
C07852=1054.448,212.979,407.658,172.141,34.905,156.536
C07853=1054.454,213.227,407.631,172.143,34.908,156.537
C07854=1054.460,213.475,407.605,172.146,34.912,156.538
C07855=1054.466,213.724,407.579,172.147,34.916,156.538
C07856=1054.473,213.973,407.553,172.149,34.920,156.539
C07857=1054.479,214.222,407.526,172.152,34.923,156.540
C07858=1054.485,214.470,407.500,172.154,34.927,156.541
C07859=1054.492,214.719,407.473,172.155,34.930,156.541
C07860=1054.498,214.967,407.447,172.157,34.934,156.542
C07861=1054.504,215.216,407.421,172.160,34.938,156.543
C07862=1054.510,215.464,407.395,172.162,34.941,156.543
C07863=1054.517,215.713,407.368,172.164,34.945,156.544
C07864=1054.523,215.961,407.342,172.165,34.949,156.545
C07865=1054.529,216.210,407.315,172.168,34.952,156.546
C07866=1054.535,216.458,407.288,172.170,34.956,156.546
C07867=1054.542,216.706,407.262,172.172,34.959,156.547
C07868=1054.548,216.956,407.236,172.174,34.963,156.548
C07869=1054.554,217.204,407.210,172.176,34.967,156.549
C07870=1054.560,217.452,407.183,172.178,34.971,156.549
C07871=1054.567,217.701,407.157,172.180,34.975,156.550
C07872=1054.573,217.950,407.130,172.182,34.978,156.551
C07873=1054.580,218.198,407.103,172.185,34.982,156.551
C07874=1054.586,218.447,407.077,172.186,34.985,156.552
C07875=1054.592,218.695,407.050,172.188,34.989,156.553
C07876=1054.599,218.944,407.024,172.190,34.993,156.554
C07877=1054.605,219.192,406.997,172.193,34.996,156.554
C07878=1054.612,219.441,406.971,172.195,34.999,156.555
C07879=1054.617,219.689,406.944,172.197,35.003,156.556
C07880=1054.623,219.938,406.917,172.198,35.006,156.556
C07881=1054.630,220.186,406.891,172.201,35.010,156.557
C07882=1054.636,220.435,406.864,172.203,35.014,156.558
C07883=1054.643,220.683,406.838,172.205,35.017,156.559
C07884=1054.649,220.927,406.811,172.207,35.021,156.559
C07885=1054.655,221.173,406.785,172.210,35.025,156.560
C07886=1054.662,221.417,406.759,172.211,35.028,156.561
C07887=1054.667,221.662,406.732,172.213,35.032,156.561
C07888=1054.674,221.906,406.706,172.215,35.035,156.562
C07889=1054.680,222.151,406.679,172.218,35.039,156.563
C07890=1054.686,222.396,406.653,172.220,35.043,156.564
C07891=1054.692,222.641,406.626,172.222,35.046,156.564
C07892=1054.699,222.888,406.600,172.223,35.050,156.565
C07893=1054.705,223.137,406.573,172.226,35.053,156.566
C07894=1054.711,223.386,406.546,172.228,35.057,156.566
C07895=1054.717,223.635,406.519,172.230,35.061,156.567
C07896=1054.723,223.883,406.492,172.233,35.064,156.568
C07897=1054.730,224.132,406.464,172.235,35.068,156.569
C07898=1054.736,224.380,406.438,172.237,35.072,156.569
C07899=1054.742,224.628,406.412,172.238,35.075,156.570
C07900=1054.749,224.877,406.384,172.241,35.079,156.571
C07901=1054.755,225.126,406.357,172.243,35.082,156.571
C07902=1054.761,225.374,406.330,172.245,35.086,156.572
C07903=1054.767,225.622,406.303,172.247,35.090,156.573
C07904=1054.773,225.871,406.276,172.250,35.093,156.574
C07905=1054.780,226.120,406.250,172.252,35.097,156.574
C07906=1054.786,226.367,406.222,172.254,35.100,156.575
C07907=1054.793,226.616,406.195,172.256,35.104,156.576
C07908=1054.799,226.865,406.169,172.259,35.107,156.576
C07909=1054.805,227.113,406.141,172.260,35.111,156.577
C07910=1054.811,227.361,406.114,172.262,35.114,156.578
C07911=1054.818,227.610,406.086,172.264,35.118,156.579
C07912=1054.825,227.859,406.060,172.267,35.121,156.579
C07913=1054.831,228.106,406.033,172.269,35.125,156.580
C07914=1054.837,228.355,406.006,172.271,35.129,156.581
C07915=1054.843,228.604,405.979,172.274,35.132,156.581
C07916=1054.850,228.852,405.951,172.276,35.136,156.582
C07917=1054.856,229.101,405.924,172.278,35.139,156.583
C07918=1054.862,229.349,405.897,172.280,35.143,156.584
C07919=1054.869,229.598,405.870,172.283,35.147,156.584
C07920=1054.875,229.846,405.843,172.285,35.150,156.585
C07921=1054.881,230.095,405.816,172.287,35.154,156.586
C07922=1054.887,230.343,405.788,172.289,35.157,156.586
C07923=1054.894,230.591,405.760,172.291,35.161,156.587
C07924=1054.900,230.840,405.733,172.293,35.165,156.588
C07925=1054.906,231.088,405.706,172.295,35.168,156.589
C07926=1054.912,231.337,405.678,172.298,35.171,156.589
C07927=1054.919,231.586,405.651,172.300,35.175,156.590
C07928=1054.925,231.833,405.623,172.302,35.178,156.591
C07929=1054.931,232.083,405.596,172.304,35.182,156.591
C07930=1054.937,232.330,405.569,172.307,35.186,156.592
C07931=1054.944,232.579,405.541,172.309,35.189,156.593
C07932=1054.950,232.828,405.514,172.311,35.193,156.594
C07933=1054.956,233.076,405.487,172.314,35.197,156.594
C07934=1054.962,233.324,405.459,172.316,35.200,156.595
C07935=1054.969,233.573,405.431,172.318,35.204,156.596
C07936=1054.975,233.821,405.404,172.320,35.207,156.596
C07937=1054.981,234.070,405.376,172.323,35.211,156.597
C07938=1054.987,234.318,405.348,172.325,35.215,156.598
C07939=1054.993,234.566,405.321,172.327,35.218,156.599
C07940=1055.000,234.807,405.294,172.330,35.222,156.599
C07941=1055.005,235.048,405.268,172.332,35.225,156.600
C07942=1055.012,235.289,405.241,172.334,35.228,156.601
C07943=1055.018,235.530,405.214,172.335,35.232,156.601
C07944=1055.024,235.770,405.188,172.338,35.235,156.602
C07945=1055.029,236.011,405.160,172.340,35.239,156.603
C07946=1055.036,236.252,405.134,172.342,35.242,156.603
C07947=1055.042,236.493,405.107,172.344,35.246,156.604
C07948=1055.048,236.741,405.079,172.347,35.249,156.605
C07949=1055.054,236.989,405.051,172.349,35.253,156.606
C07950=1055.061,237.238,405.024,172.351,35.256,156.606
C07951=1055.067,237.486,404.995,172.354,35.260,156.607
C07952=1055.074,237.735,404.968,172.356,35.264,156.608
C07953=1055.080,237.982,404.940,172.358,35.267,156.608
C07954=1055.086,238.231,404.912,172.360,35.271,156.609
C07955=1055.092,238.480,404.884,172.363,35.274,156.610
C07956=1055.099,238.729,404.857,172.365,35.277,156.611
C07957=1055.106,238.977,404.830,172.367,35.281,156.611
C07958=1055.111,239.225,404.802,172.370,35.285,156.612
C07959=1055.118,239.473,404.773,172.372,35.288,156.613
C07960=1055.125,239.721,404.745,172.375,35.292,156.613
C07961=1055.130,239.970,404.717,172.377,35.295,156.614
C07962=1055.137,240.218,404.690,172.380,35.299,156.615
C07963=1055.143,240.466,404.662,172.382,35.303,156.616
C07964=1055.149,240.715,404.634,172.384,35.306,156.616
C07965=1055.156,240.964,404.606,172.387,35.310,156.617
C07966=1055.162,241.212,404.578,172.389,35.313,156.618
C07967=1055.168,241.461,404.550,172.391,35.316,156.618
C07968=1055.175,241.709,404.523,172.394,35.320,156.619
C07969=1055.181,241.957,404.494,172.396,35.324,156.620
C07970=1055.187,242.206,404.466,172.398,35.327,156.621
C07971=1055.193,242.454,404.437,172.400,35.331,156.621
C07972=1055.200,242.702,404.410,172.403,35.334,156.622
C07973=1055.205,242.950,404.382,172.405,35.338,156.623
C07974=1055.211,243.199,404.353,172.407,35.341,156.623
C07975=1055.218,243.447,404.325,172.410,35.345,156.624
C07976=1055.224,243.696,404.297,172.412,35.349,156.625
C07977=1055.231,243.944,404.269,172.415,35.352,156.626
C07978=1055.237,244.193,404.241,172.418,35.356,156.626
C07979=1055.243,244.440,404.213,172.420,35.359,156.627
C07980=1055.249,244.689,404.184,172.422,35.363,156.628
C07981=1055.255,244.937,404.156,172.424,35.367,156.629
C07982=1055.262,245.185,404.127,172.427,35.370,156.629
C07983=1055.268,245.434,404.099,172.429,35.373,156.630
C07984=1055.275,245.683,404.071,172.431,35.377,156.631
C07985=1055.281,245.931,404.042,172.434,35.380,156.631
C07986=1055.287,246.179,404.014,172.436,35.384,156.632
C07987=1055.293,246.427,403.987,172.438,35.387,156.633
C07988=1055.299,246.675,403.958,172.442,35.391,156.634
C07989=1055.305,246.924,403.929,172.444,35.395,156.634
C07990=1055.312,247.172,403.900,172.446,35.398,156.635
C07991=1055.318,247.421,403.872,172.448,35.402,156.636
C07992=1055.324,247.669,403.843,172.451,35.405,156.636
C07993=1055.330,247.917,403.815,172.453,35.409,156.637
C07994=1055.336,248.165,403.786,172.455,35.413,156.638
C07995=1055.342,248.414,403.758,172.458,35.417,156.639
C07996=1055.348,248.652,403.731,172.460,35.420,156.639
C07997=1055.354,248.889,403.703,172.462,35.423,156.640
C07998=1055.360,249.127,403.675,172.465,35.427,156.641
C07999=1055.366,249.365,403.648,172.467,35.430,156.642
C08000=1055.371,249.602,403.621,172.469,35.433,156.642
C08001=1055.377,249.841,403.594,172.472,35.437,156.643
C08002=1055.384,250.078,403.566,172.475,35.441,156.644
C08003=1055.390,250.316,403.539,172.477,35.444,156.644
C08004=1055.396,250.564,403.510,172.479,35.447,156.645
C08005=1055.402,250.813,403.481,172.482,35.451,156.646
C08006=1055.408,251.061,403.452,172.484,35.454,156.646
C08007=1055.415,251.309,403.424,172.486,35.458,156.647
C08008=1055.421,251.558,403.395,172.489,35.461,156.648
C08009=1055.427,251.806,403.366,172.492,35.465,156.649
C08010=1055.434,252.054,403.337,172.494,35.469,156.649
C08011=1055.439,252.303,403.309,172.497,35.472,156.650
C08012=1055.446,252.551,403.280,172.499,35.476,156.651
C08013=1055.452,252.799,403.251,172.501,35.479,156.652
C08014=1055.458,253.048,403.223,172.504,35.483,156.652
C08015=1055.465,253.295,403.194,172.507,35.487,156.653
C08016=1055.471,253.544,403.165,172.509,35.490,156.654
C08017=1055.477,253.792,403.136,172.512,35.494,156.654
C08018=1055.484,254.040,403.107,172.514,35.497,156.655
C08019=1055.490,254.289,403.079,172.516,35.501,156.656
C08020=1055.496,254.537,403.050,172.519,35.504,156.657
C08021=1055.502,254.785,403.021,172.522,35.508,156.657
C08022=1055.508,255.033,402.992,172.524,35.512,156.658
C08023=1055.515,255.281,402.963,172.526,35.515,156.659
C08024=1055.521,255.529,402.934,172.529,35.519,156.660
C08025=1055.527,255.778,402.905,172.532,35.522,156.660
C08026=1055.534,256.026,402.876,172.534,35.525,156.661
C08027=1055.541,256.275,402.847,172.537,35.529,156.662
C08028=1055.547,256.523,402.818,172.539,35.532,156.662
C08029=1055.553,256.771,402.789,172.541,35.536,156.663
C08030=1055.559,257.019,402.760,172.545,35.539,156.664
C08031=1055.566,257.267,402.731,172.547,35.543,156.665
C08032=1055.572,257.515,402.702,172.549,35.547,156.665
C08033=1055.578,257.763,402.673,172.552,35.550,156.666
C08034=1055.585,258.012,402.644,172.555,35.554,156.667
C08035=1055.591,258.260,402.615,172.557,35.557,156.668
C08036=1055.597,258.509,402.586,172.560,35.560,156.668
C08037=1055.604,258.757,402.557,172.562,35.564,156.669
C08038=1055.610,259.005,402.528,172.565,35.567,156.670
C08039=1055.617,259.254,402.498,172.568,35.571,156.670
C08040=1055.623,259.502,402.469,172.570,35.575,156.671
C08041=1055.630,259.750,402.441,172.572,35.578,156.672
C08042=1055.636,259.998,402.412,172.576,35.582,156.673
C08043=1055.643,260.246,402.383,172.578,35.585,156.673
C08044=1055.649,260.495,402.353,172.580,35.588,156.674
C08045=1055.656,260.742,402.323,172.584,35.592,156.675
C08046=1055.662,260.990,402.294,172.586,35.595,156.675
C08047=1055.668,261.238,402.265,172.588,35.599,156.676
C08048=1055.675,261.487,402.236,172.591,35.602,156.677
C08049=1055.682,261.735,402.207,172.594,35.606,156.678
C08050=1055.688,261.984,402.178,172.596,35.610,156.678
C08051=1055.694,262.232,402.149,172.599,35.613,156.679
C08052=1055.701,262.468,402.120,172.602,35.616,156.680
C08053=1055.707,262.706,402.092,172.604,35.620,156.680
C08054=1055.713,262.943,402.064,172.606,35.623,156.681
C08055=1055.719,263.179,402.036,172.609,35.626,156.682
C08056=1055.725,263.416,402.008,172.611,35.630,156.682
C08057=1055.731,263.652,401.980,172.614,35.633,156.683
C08058=1055.737,263.889,401.952,172.617,35.636,156.684
C08059=1055.743,264.126,401.924,172.619,35.640,156.685
C08060=1055.750,264.374,401.894,172.621,35.643,156.685
C08061=1055.755,264.623,401.864,172.625,35.647,156.686
C08062=1055.762,264.870,401.834,172.627,35.651,156.687
C08063=1055.768,265.118,401.805,172.629,35.654,156.688
C08064=1055.774,265.368,401.775,172.633,35.658,156.688
C08065=1055.781,265.615,401.746,172.635,35.661,156.689
C08066=1055.787,265.863,401.717,172.637,35.665,156.690
C08067=1055.793,266.111,401.686,172.641,35.668,156.690
C08068=1055.800,266.360,401.657,172.643,35.672,156.691
C08069=1055.806,266.607,401.627,172.646,35.675,156.692
C08070=1055.812,266.856,401.597,172.649,35.679,156.693
C08071=1055.819,267.104,401.567,172.651,35.683,156.693
C08072=1055.825,267.352,401.538,172.654,35.686,156.694
C08073=1055.831,267.600,401.508,172.657,35.690,156.695
C08074=1055.838,267.849,401.479,172.659,35.693,156.696
C08075=1055.844,268.097,401.448,172.662,35.697,156.696
C08076=1055.850,268.345,401.419,172.665,35.700,156.697
C08077=1055.857,268.593,401.389,172.667,35.704,156.698
C08078=1055.863,268.841,401.359,172.670,35.707,156.699
C08079=1055.869,269.089,401.330,172.673,35.711,156.699
C08080=1055.876,269.338,401.299,172.675,35.714,156.700
C08081=1055.882,269.585,401.269,172.678,35.718,156.701
C08082=1055.888,269.834,401.239,172.681,35.722,156.702
C08083=1055.895,270.082,401.209,172.683,35.726,156.702
C08084=1055.901,270.330,401.179,172.687,35.729,156.703
C08085=1055.907,270.578,401.150,172.689,35.733,156.704
C08086=1055.913,270.826,401.119,172.692,35.736,156.705
C08087=1055.920,271.074,401.090,172.695,35.740,156.705
C08088=1055.926,271.322,401.059,172.697,35.743,156.706
C08089=1055.932,271.570,401.030,172.701,35.747,156.707
C08090=1055.939,271.819,400.999,172.703,35.751,156.708
C08091=1055.945,272.066,400.969,172.705,35.754,156.708
C08092=1055.952,272.315,400.939,172.709,35.758,156.709
C08093=1055.958,272.562,400.909,172.711,35.761,156.710
C08094=1055.964,272.811,400.879,172.714,35.765,156.711
C08095=1055.970,273.059,400.849,172.717,35.768,156.711
C08096=1055.977,273.307,400.819,172.719,35.772,156.712
C08097=1055.983,273.555,400.788,172.722,35.776,156.713
C08098=1055.989,273.803,400.758,172.725,35.779,156.714
C08099=1055.996,274.051,400.728,172.728,35.783,156.714
C08100=1056.002,274.299,400.697,172.731,35.787,156.715
C08101=1056.008,274.547,400.667,172.733,35.790,156.716
C08102=1056.015,274.795,400.637,172.736,35.794,156.717
C08103=1056.021,275.043,400.606,172.739,35.797,156.717
C08104=1056.027,275.292,400.576,172.742,35.801,156.718
C08105=1056.034,275.539,400.546,172.744,35.804,156.719
C08106=1056.040,275.788,400.515,172.748,35.808,156.720
C08107=1056.046,276.035,400.485,172.750,35.812,156.720
C08108=1056.053,276.275,400.456,172.753,35.815,156.721
C08109=1056.059,276.513,400.427,172.756,35.818,156.722
C08110=1056.064,276.752,400.397,172.758,35.822,156.723
C08111=1056.071,276.991,400.368,172.761,35.825,156.723
C08112=1056.077,277.229,400.339,172.764,35.829,156.724
C08113=1056.083,277.468,400.309,172.766,35.832,156.725
C08114=1056.089,277.707,400.280,172.770,35.836,156.726
C08115=1056.095,277.946,400.251,172.772,35.840,156.726
C08116=1056.102,278.194,400.220,172.774,35.843,156.727
C08117=1056.108,278.442,400.190,172.778,35.847,156.728
C08118=1056.114,278.690,400.158,172.780,35.850,156.729
C08119=1056.121,278.939,400.128,172.784,35.854,156.729
C08120=1056.127,279.186,400.098,172.786,35.858,156.730
C08121=1056.134,279.435,400.067,172.789,35.861,156.731
C08122=1056.140,279.682,400.037,172.792,35.865,156.732
C08123=1056.146,279.930,400.005,172.795,35.868,156.732
C08124=1056.152,280.178,399.975,172.797,35.872,156.733
C08125=1056.159,280.427,399.944,172.801,35.876,156.734
C08126=1056.165,280.675,399.913,172.803,35.880,156.735
C08127=1056.171,280.922,399.882,172.807,35.883,156.735
C08128=1056.177,281.171,399.852,172.809,35.887,156.736
C08129=1056.184,281.418,399.821,172.812,35.891,156.737
C08130=1056.190,281.667,399.790,172.815,35.894,156.738
C08131=1056.197,281.915,399.758,172.818,35.898,156.739
C08132=1056.203,282.162,399.728,172.821,35.901,156.739
C08133=1056.209,282.411,399.697,172.824,35.905,156.740
C08134=1056.215,282.658,399.666,172.826,35.909,156.741
C08135=1056.222,282.907,399.636,172.830,35.912,156.742
C08136=1056.228,283.154,399.604,172.832,35.916,156.742
C08137=1056.234,283.402,399.574,172.836,35.920,156.743
C08138=1056.241,283.650,399.542,172.838,35.924,156.744
C08139=1056.247,283.899,399.512,172.841,35.927,156.745
C08140=1056.253,284.146,399.481,172.845,35.931,156.746
C08141=1056.260,284.394,399.450,172.847,35.935,156.746
C08142=1056.266,284.642,399.418,172.851,35.938,156.747
C08143=1056.272,284.890,399.388,172.853,35.942,156.748
C08144=1056.279,285.138,399.357,172.856,35.945,156.749
C08145=1056.286,285.386,399.325,172.859,35.949,156.750
C08146=1056.292,285.634,399.295,172.862,35.953,156.750
C08147=1056.298,285.882,399.263,172.864,35.956,156.751
C08148=1056.305,286.130,399.232,172.868,35.960,156.752
C08149=1056.311,286.378,399.201,172.871,35.964,156.753
C08150=1056.318,286.625,399.170,172.874,35.968,156.753
C08151=1056.324,286.873,399.139,172.877,35.971,156.754
C08152=1056.331,287.122,399.108,172.879,35.975,156.755
C08153=1056.337,287.370,399.077,172.883,35.979,156.756
C08154=1056.344,287.617,399.046,172.886,35.982,156.757
C08155=1056.350,287.865,399.015,172.889,35.986,156.757
C08156=1056.356,288.114,398.983,172.892,35.989,156.758
C08157=1056.363,288.361,398.951,172.895,35.993,156.759
C08158=1056.369,288.609,398.920,172.898,35.997,156.760
C08159=1056.376,288.857,398.889,172.900,36.000,156.760
C08160=1056.381,289.105,398.858,172.904,36.004,156.761
C08161=1056.388,289.353,398.826,172.907,36.008,156.762
C08162=1056.395,289.601,398.795,172.910,36.011,156.763
C08163=1056.401,289.848,398.764,172.913,36.016,156.764
C08164=1056.407,290.093,398.733,172.915,36.019,156.764
C08165=1056.413,290.337,398.701,172.919,36.023,156.765
C08166=1056.420,290.581,398.670,172.922,36.027,156.766
C08167=1056.426,290.826,398.640,172.925,36.030,156.767
C08168=1056.432,291.070,398.609,172.928,36.034,156.768
C08169=1056.438,291.314,398.577,172.931,36.038,156.768
C08170=1056.445,291.559,398.546,172.934,36.041,156.769
C08171=1056.451,291.803,398.515,172.937,36.045,156.770
C08172=1056.457,292.051,398.484,172.940,36.049,156.771
C08173=1056.463,292.299,398.452,172.943,36.052,156.772
C08174=1056.470,292.547,398.420,172.947,36.056,156.772
C08175=1056.477,292.795,398.389,172.949,36.060,156.773
C08176=1056.483,293.043,398.357,172.952,36.063,156.774
C08177=1056.490,293.291,398.325,172.956,36.068,156.775
C08178=1056.497,293.538,398.293,172.958,36.071,156.776
C08179=1056.503,293.786,398.261,172.962,36.075,156.776
C08180=1056.509,294.033,398.230,172.965,36.079,156.777
C08181=1056.515,294.281,398.199,172.968,36.082,156.778
C08182=1056.521,294.529,398.167,172.971,36.086,156.779
C08183=1056.528,294.777,398.135,172.974,36.090,156.780
C08184=1056.534,295.025,398.102,172.977,36.094,156.780
C08185=1056.541,295.273,398.071,172.980,36.097,156.781
C08186=1056.547,295.521,398.039,172.984,36.101,156.782
C08187=1056.554,295.769,398.008,172.986,36.105,156.783
C08188=1056.560,296.017,397.975,172.990,36.109,156.784
C08189=1056.567,296.265,397.943,172.993,36.112,156.784
C08190=1056.573,296.513,397.911,172.996,36.116,156.785
C08191=1056.580,296.761,397.880,172.999,36.120,156.786
C08192=1056.586,297.008,397.847,173.002,36.124,156.787
C08193=1056.592,297.256,397.815,173.005,36.128,156.788
C08194=1056.598,297.503,397.783,173.008,36.132,156.789
C08195=1056.604,297.751,397.751,173.012,36.136,156.790
C08196=1056.611,297.999,397.719,173.015,36.140,156.790
C08197=1056.617,298.247,397.687,173.018,36.143,156.791
C08198=1056.624,298.494,397.654,173.021,36.147,156.792
C08199=1056.630,298.743,397.622,173.025,36.151,156.793
C08200=1056.636,298.990,397.590,173.027,36.155,156.794
C08201=1056.642,299.238,397.558,173.030,36.159,156.795
C08202=1056.648,299.486,397.525,173.034,36.163,156.795
C08203=1056.655,299.734,397.493,173.036,36.166,156.796
C08204=1056.661,299.981,397.461,173.040,36.171,156.797
C08205=1056.667,300.230,397.429,173.043,36.175,156.798
C08206=1056.674,300.477,397.396,173.047,36.178,156.799
C08207=1056.680,300.725,397.363,173.049,36.182,156.800
C08208=1056.687,300.973,397.332,173.053,36.186,156.801
C08209=1056.693,301.220,397.299,173.056,36.190,156.801
C08210=1056.699,301.468,397.266,173.060,36.194,156.802
C08211=1056.705,301.716,397.234,173.062,36.198,156.803
C08212=1056.711,301.964,397.201,173.066,36.202,156.804
C08213=1056.718,302.211,397.169,173.069,36.205,156.805
C08214=1056.724,302.459,397.137,173.072,36.209,156.806
C08215=1056.731,302.707,397.105,173.076,36.213,156.806
C08216=1056.737,302.954,397.072,173.078,36.217,156.807
C08217=1056.744,303.203,397.039,173.082,36.221,156.808
C08218=1056.750,303.451,397.007,173.085,36.225,156.809
C08219=1056.757,303.698,396.975,173.089,36.229,156.810
C08220=1056.764,303.955,396.941,173.092,36.233,156.811
C08221=1056.769,304.210,396.907,173.095,36.237,156.812
C08222=1056.776,304.467,396.873,173.098,36.241,156.813
C08223=1056.783,304.724,396.839,173.102,36.245,156.813
C08224=1056.789,304.971,396.807,173.105,36.249,156.814
C08225=1056.796,305.219,396.775,173.109,36.253,156.815
C08226=1056.803,305.467,396.741,173.112,36.257,156.816
C08227=1056.809,305.715,396.709,173.116,36.261,156.817
C08228=1056.816,305.962,396.676,173.118,36.264,156.818
C08229=1056.822,306.210,396.643,173.122,36.268,156.818
C08230=1056.828,306.457,396.611,173.125,36.273,156.819
C08231=1056.835,306.706,396.577,173.129,36.277,156.820
C08232=1056.842,306.953,396.545,173.132,36.280,156.821
C08233=1056.848,307.200,396.513,173.136,36.284,156.822
C08234=1056.855,307.448,396.480,173.138,36.288,156.823
C08235=1056.862,307.696,396.447,173.142,36.292,156.824
C08236=1056.868,307.944,396.414,173.145,36.296,156.825
C08237=1056.874,308.192,396.381,173.149,36.300,156.825
C08238=1056.880,308.439,396.348,173.152,36.304,156.826
C08239=1056.887,308.687,396.315,173.156,36.308,156.827
C08240=1056.894,308.935,396.283,173.159,36.312,156.828
C08241=1056.901,309.182,396.250,173.163,36.316,156.829
C08242=1056.908,309.430,396.217,173.165,36.320,156.830
C08243=1056.914,309.678,396.184,173.168,36.323,156.831
C08244=1056.920,309.925,396.151,173.172,36.327,156.831
C08245=1056.927,310.173,396.118,173.176,36.331,156.832
C08246=1056.934,310.421,396.085,173.179,36.335,156.833
C08247=1056.940,310.668,396.052,173.183,36.340,156.834
C08248=1056.947,310.916,396.019,173.186,36.344,156.835
C08249=1056.953,311.164,395.986,173.189,36.347,156.836
C08250=1056.960,311.412,395.953,173.193,36.351,156.837
C08251=1056.967,311.659,395.919,173.196,36.355,156.838
C08252=1056.973,311.907,395.887,173.199,36.359,156.838
C08253=1056.980,312.155,395.854,173.203,36.363,156.839
C08254=1056.987,312.402,395.820,173.206,36.367,156.840
C08255=1056.994,312.650,395.787,173.210,36.371,156.841
C08256=1057.000,312.898,395.754,173.213,36.375,156.842
C08257=1057.008,313.145,395.721,173.216,36.379,156.843
C08258=1057.014,313.393,395.688,173.220,36.383,156.844
C08259=1057.020,313.642,395.655,173.224,36.387,156.845
C08260=1057.027,313.888,395.621,173.227,36.391,156.846
C08261=1057.033,314.136,395.587,173.231,36.395,156.847
C08262=1057.040,314.384,395.554,173.234,36.399,156.847
C08263=1057.046,314.631,395.520,173.238,36.403,156.848
C08264=1057.052,314.879,395.487,173.241,36.407,156.849
C08265=1057.058,315.127,395.453,173.245,36.412,156.850
C08266=1057.065,315.374,395.419,173.247,36.416,156.851
C08267=1057.071,315.621,395.387,173.251,36.420,156.852
C08268=1057.078,315.869,395.352,173.254,36.424,156.853
C08269=1057.084,316.117,395.319,173.258,36.428,156.854
C08270=1057.090,316.365,395.285,173.261,36.433,156.855
C08271=1057.097,316.612,395.251,173.265,36.437,156.856
C08272=1057.103,316.860,395.217,173.269,36.441,156.857
C08273=1057.110,317.108,395.184,173.272,36.445,156.858
C08274=1057.116,317.356,395.150,173.276,36.449,156.859
C08275=1057.123,317.603,395.116,173.279,36.453,156.859
C08276=1057.129,317.864,395.080,173.283,36.458,156.860
C08277=1057.136,318.124,395.045,173.286,36.462,156.861
C08278=1057.143,318.385,395.009,173.290,36.467,156.862
C08279=1057.149,318.645,394.974,173.295,36.471,156.863
C08280=1057.157,318.892,394.940,173.298,36.475,156.864
C08281=1057.163,319.140,394.906,173.302,36.479,156.865
C08282=1057.169,319.388,394.872,173.305,36.483,156.866
C08283=1057.176,319.635,394.838,173.309,36.488,156.867
C08284=1057.182,319.883,394.805,173.312,36.492,156.868
C08285=1057.189,320.131,394.771,173.316,36.496,156.869
C08286=1057.195,320.378,394.737,173.319,36.500,156.870
C08287=1057.202,320.626,394.703,173.323,36.504,156.871
C08288=1057.208,320.873,394.669,173.326,36.508,156.872
C08289=1057.215,321.121,394.635,173.330,36.513,156.873
C08290=1057.222,321.369,394.601,173.334,36.517,156.874
C08291=1057.228,321.616,394.567,173.337,36.521,156.875
C08292=1057.235,321.864,394.533,173.341,36.526,156.876
C08293=1057.241,322.112,394.498,173.344,36.530,156.877
C08294=1057.248,322.359,394.465,173.348,36.534,156.878
C08295=1057.254,322.606,394.430,173.351,36.538,156.878
C08296=1057.262,322.854,394.396,173.355,36.542,156.879
C08297=1057.268,323.101,394.362,173.359,36.547,156.880
C08298=1057.274,323.349,394.328,173.362,36.551,156.881
C08299=1057.281,323.597,394.294,173.366,36.555,156.882
C08300=1057.288,323.845,394.259,173.369,36.559,156.883
C08301=1057.294,324.092,394.226,173.373,36.563,156.884
C08302=1057.301,324.339,394.191,173.376,36.568,156.885
C08303=1057.308,324.587,394.157,173.380,36.572,156.886
C08304=1057.315,324.835,394.122,173.385,36.576,156.887
C08305=1057.321,325.082,394.088,173.388,36.580,156.888
C08306=1057.328,325.329,394.054,173.392,36.585,156.889
C08307=1057.334,325.577,394.019,173.395,36.589,156.890
C08308=1057.341,325.825,393.985,173.399,36.594,156.891
C08309=1057.348,326.073,393.951,173.403,36.598,156.892
C08310=1057.354,326.319,393.916,173.406,36.602,156.893
C08311=1057.362,326.567,393.883,173.410,36.606,156.894
C08312=1057.368,326.815,393.848,173.413,36.611,156.895
C08313=1057.375,327.062,393.813,173.418,36.615,156.896
C08314=1057.382,327.310,393.779,173.422,36.619,156.897
C08315=1057.389,327.558,393.744,173.425,36.623,156.898
C08316=1057.395,327.805,393.710,173.429,36.628,156.899
C08317=1057.403,328.053,393.675,173.432,36.632,156.900
C08318=1057.409,328.300,393.641,173.436,36.636,156.901
C08319=1057.415,328.547,393.606,173.441,36.641,156.902
C08320=1057.423,328.795,393.572,173.444,36.645,156.903
C08321=1057.429,329.042,393.537,173.448,36.649,156.904
C08322=1057.436,329.290,393.503,173.451,36.653,156.905
C08323=1057.443,329.537,393.468,173.455,36.658,156.906
C08324=1057.450,329.785,393.434,173.459,36.662,156.907
C08325=1057.456,330.033,393.398,173.463,36.666,156.908
C08326=1057.464,330.280,393.365,173.467,36.671,156.909
C08327=1057.470,330.528,393.329,173.470,36.676,156.910
C08328=1057.477,330.775,393.294,173.474,36.680,156.911
C08329=1057.483,331.023,393.259,173.478,36.684,156.912
C08330=1057.490,331.271,393.224,173.481,36.689,156.913
C08331=1057.496,331.518,393.189,173.486,36.693,156.914
C08332=1057.503,331.773,393.153,173.490,36.698,156.915
C08333=1057.511,332.028,393.117,173.493,36.702,156.916
C08334=1057.518,332.283,393.081,173.498,36.707,156.917
C08335=1057.524,332.538,393.046,173.502,36.712,156.918
C08336=1057.531,332.785,393.011,173.505,36.716,156.919
C08337=1057.538,333.033,392.975,173.509,36.721,156.920
C08338=1057.544,333.280,392.940,173.513,36.725,156.921
C08339=1057.550,333.528,392.905,173.517,36.729,156.922
C08340=1057.557,333.775,392.869,173.521,36.734,156.923
C08341=1057.564,334.023,392.834,173.524,36.738,156.924
C08342=1057.571,334.271,392.799,173.528,36.743,156.925
C08343=1057.578,334.518,392.764,173.533,36.748,156.926
C08344=1057.585,334.765,392.729,173.536,36.752,156.927
C08345=1057.592,335.013,392.693,173.540,36.757,156.928
C08346=1057.598,335.260,392.658,173.544,36.761,156.929
C08347=1057.605,335.507,392.623,173.548,36.766,156.930
C08348=1057.612,335.755,392.588,173.552,36.770,156.931
C08349=1057.619,336.002,392.553,173.556,36.775,156.932
C08350=1057.625,336.250,392.517,173.559,36.780,156.934
C08351=1057.631,336.497,392.482,173.564,36.784,156.935
C08352=1057.639,336.745,392.446,173.568,36.789,156.936
C08353=1057.646,336.992,392.411,173.571,36.793,156.937
C08354=1057.653,337.239,392.376,173.576,36.798,156.938
C08355=1057.659,337.487,392.340,173.580,36.802,156.939
C08356=1057.665,337.734,392.305,173.583,36.807,156.940
C08357=1057.672,337.981,392.269,173.587,36.812,156.941
C08358=1057.679,338.229,392.233,173.592,36.817,156.942
C08359=1057.685,338.476,392.198,173.596,36.821,156.943
C08360=1057.693,338.724,392.162,173.599,36.826,156.944
C08361=1057.699,338.971,392.126,173.604,36.831,156.945
C08362=1057.706,339.219,392.091,173.608,36.835,156.946
C08363=1057.713,339.465,392.055,173.611,36.840,156.947
C08364=1057.719,339.713,392.019,173.616,36.845,156.949
C08365=1057.726,339.961,391.984,173.620,36.849,156.950
C08366=1057.733,340.208,391.948,173.623,36.854,156.951
C08367=1057.739,340.456,391.912,173.628,36.859,156.952
C08368=1057.746,340.702,391.876,173.632,36.863,156.953
C08369=1057.754,340.950,391.841,173.636,36.868,156.954
C08370=1057.760,341.197,391.804,173.640,36.873,156.955
C08371=1057.767,341.445,391.769,173.644,36.877,156.956
C08372=1057.773,341.692,391.733,173.648,36.882,156.957
C08373=1057.781,341.939,391.697,173.652,36.887,156.958
C08374=1057.788,342.187,391.661,173.656,36.892,156.959
C08375=1057.794,342.434,391.625,173.661,36.897,156.961
C08376=1057.801,342.682,391.590,173.665,36.901,156.962
C08377=1057.808,342.929,391.554,173.668,36.906,156.963
C08378=1057.815,343.176,391.517,173.673,36.911,156.964
C08379=1057.822,343.424,391.482,173.677,36.916,156.965
C08380=1057.828,343.671,391.445,173.680,36.920,156.966
C08381=1057.835,343.918,391.409,173.685,36.925,156.967
C08382=1057.842,344.165,391.373,173.689,36.930,156.969
C08383=1057.849,344.413,391.337,173.694,36.935,156.970
C08384=1057.856,344.660,391.301,173.697,36.940,156.971
C08385=1057.863,344.907,391.264,173.701,36.944,156.972
C08386=1057.869,345.154,391.228,173.706,36.949,156.973
C08387=1057.877,345.402,391.192,173.710,36.954,156.974
C08388=1057.883,345.653,391.155,173.715,36.960,156.975
C08389=1057.890,345.903,391.118,173.718,36.964,156.976
C08390=1057.897,346.154,391.081,173.723,36.969,156.978
C08391=1057.904,346.405,391.045,173.727,36.974,156.979
C08392=1057.911,346.653,391.008,173.732,36.979,156.980
C08393=1057.918,346.899,390.972,173.735,36.984,156.981
C08394=1057.925,347.147,390.935,173.740,36.989,156.982
C08395=1057.931,347.394,390.899,173.744,36.994,156.983
C08396=1057.938,347.642,390.862,173.748,36.999,156.985
C08397=1057.945,347.888,390.825,173.752,37.004,156.986
C08398=1057.952,348.135,390.789,173.756,37.009,156.987
C08399=1057.959,348.383,390.752,173.761,37.014,156.988
C08400=1057.966,348.630,390.716,173.765,37.019,156.989
C08401=1057.973,348.877,390.680,173.770,37.024,156.991
C08402=1057.979,349.125,390.643,173.773,37.028,156.992
C08403=1057.986,349.372,390.606,173.778,37.033,156.993
C08404=1057.994,349.619,390.569,173.782,37.039,156.994
C08405=1058.000,349.866,390.533,173.787,37.044,156.995
C08406=1058.007,350.114,390.496,173.790,37.049,156.996
C08407=1058.014,350.360,390.459,173.795,37.054,156.998
C08408=1058.021,350.608,390.423,173.799,37.059,156.999
C08409=1058.028,350.856,390.386,173.804,37.064,157.000
C08410=1058.035,351.103,390.349,173.809,37.069,157.001
C08411=1058.042,351.350,390.312,173.813,37.074,157.002
C08412=1058.048,351.597,390.275,173.817,37.079,157.004
C08413=1058.055,351.844,390.238,173.821,37.084,157.005
C08414=1058.063,352.091,390.202,173.826,37.089,157.006
C08415=1058.070,352.338,390.165,173.830,37.094,157.007
C08416=1058.077,352.586,390.128,173.835,37.099,157.008
C08417=1058.083,352.832,390.091,173.839,37.105,157.010
C08418=1058.090,353.080,390.054,173.843,37.110,157.011
C08419=1058.098,353.327,390.016,173.847,37.115,157.012
C08420=1058.104,353.574,389.980,173.852,37.120,157.013
C08421=1058.111,353.821,389.942,173.857,37.126,157.015
C08422=1058.118,354.068,389.905,173.861,37.131,157.016
C08423=1058.125,354.315,389.868,173.866,37.136,157.017
C08424=1058.132,354.562,389.831,173.869,37.141,157.018
C08425=1058.139,354.809,389.793,173.874,37.146,157.020
C08426=1058.146,355.057,389.756,173.879,37.151,157.021
C08427=1058.153,355.304,389.719,173.883,37.157,157.022
C08428=1058.160,355.551,389.682,173.888,37.162,157.023
C08429=1058.167,355.798,389.644,173.892,37.167,157.025
C08430=1058.175,356.045,389.607,173.897,37.172,157.026
C08431=1058.181,356.292,389.570,173.901,37.177,157.027
C08432=1058.188,356.539,389.533,173.905,37.183,157.028
C08433=1058.195,356.786,389.495,173.910,37.188,157.030
C08434=1058.203,357.034,389.458,173.915,37.193,157.031
C08435=1058.209,357.281,389.420,173.919,37.198,157.032
C08436=1058.216,357.527,389.382,173.924,37.204,157.033
C08437=1058.223,357.775,389.345,173.929,37.210,157.035
C08438=1058.230,358.022,389.307,173.933,37.215,157.036
C08439=1058.237,358.269,389.270,173.937,37.220,157.037
C08440=1058.245,358.516,389.232,173.942,37.225,157.039
C08441=1058.252,358.763,389.195,173.946,37.231,157.040
C08442=1058.258,359.010,389.157,173.951,37.236,157.041
C08443=1058.265,359.257,389.119,173.956,37.242,157.043
C08444=1058.277,359.666,389.057,173.964,37.251,157.045
C08445=1058.288,360.074,388.995,173.971,37.259,157.047
C08446=1058.301,360.482,388.932,173.979,37.268,157.049
C08447=1058.312,360.891,388.869,173.986,37.277,157.051
C08448=1058.319,361.138,388.832,173.991,37.283,157.052
C08449=1058.326,361.384,388.794,173.995,37.288,157.054
C08450=1058.334,361.631,388.756,174.000,37.294,157.055
C08451=1058.340,361.879,388.718,174.005,37.299,157.056
C08452=1058.348,362.125,388.680,174.010,37.305,157.058
C08453=1058.355,362.372,388.643,174.014,37.310,157.059
C08454=1058.362,362.619,388.604,174.019,37.316,157.060
C08455=1058.369,362.866,388.566,174.024,37.321,157.062
C08456=1058.376,363.113,388.528,174.029,37.327,157.063
C08457=1058.384,363.361,388.489,174.034,37.333,157.064
C08458=1058.391,363.608,388.452,174.038,37.338,157.066
C08459=1058.398,363.855,388.414,174.042,37.344,157.067
C08460=1058.405,364.101,388.375,174.048,37.350,157.069
C08461=1058.412,364.349,388.337,174.053,37.355,157.070
C08462=1058.419,364.595,388.298,174.056,37.361,157.071
C08463=1058.427,364.842,388.260,174.061,37.366,157.073
C08464=1058.433,365.089,388.222,174.066,37.372,157.074
C08465=1058.440,365.336,388.183,174.071,37.378,157.075
C08466=1058.448,365.583,388.145,174.076,37.383,157.077
C08467=1058.454,365.830,388.107,174.080,37.389,157.078
C08468=1058.462,366.077,388.069,174.085,37.395,157.080
C08469=1058.469,366.323,388.030,174.091,37.401,157.081
C08470=1058.476,366.570,387.992,174.095,37.406,157.082
C08471=1058.484,366.817,387.952,174.100,37.412,157.084
C08472=1058.490,367.064,387.914,174.106,37.418,157.085
C08473=1058.498,367.311,387.876,174.109,37.424,157.087
C08474=1058.504,367.558,387.837,174.115,37.430,157.088
C08475=1058.512,367.805,387.799,174.120,37.435,157.090
C08476=1058.522,368.145,387.745,174.126,37.443,157.092
C08477=1058.532,368.487,387.691,174.133,37.452,157.094
C08478=1058.541,368.828,387.638,174.140,37.459,157.095
C08479=1058.551,369.168,387.584,174.147,37.467,157.097
C08480=1058.560,369.416,387.546,174.151,37.474,157.099
C08481=1058.566,369.663,387.507,174.156,37.479,157.100
C08482=1058.573,369.909,387.468,174.161,37.485,157.102
C08483=1058.581,370.157,387.429,174.167,37.491,157.103
C08484=1058.588,370.403,387.391,174.172,37.497,157.105
C08485=1058.595,370.650,387.352,174.177,37.503,157.106
C08486=1058.603,370.896,387.313,174.182,37.509,157.108
C08487=1058.610,371.144,387.274,174.187,37.515,157.109
C08488=1058.618,371.390,387.235,174.192,37.521,157.111
C08489=1058.626,371.637,387.195,174.197,37.526,157.112
C08490=1058.632,371.884,387.157,174.202,37.532,157.113
C08491=1058.640,372.130,387.118,174.207,37.538,157.115
C08492=1058.648,372.377,387.078,174.212,37.544,157.116
C08493=1058.654,372.624,387.040,174.217,37.550,157.118
C08494=1058.662,372.870,387.000,174.222,37.556,157.119
C08495=1058.669,373.118,386.961,174.228,37.562,157.121
C08496=1058.677,373.392,386.917,174.233,37.569,157.123
C08497=1058.685,373.665,386.873,174.238,37.576,157.124
C08498=1058.692,373.940,386.830,174.244,37.583,157.126
C08499=1058.701,374.214,386.786,174.250,37.590,157.128
C08500=1058.709,374.460,386.747,174.255,37.596,157.129
C08501=1058.716,374.707,386.707,174.260,37.602,157.131
C08502=1058.723,374.953,386.668,174.265,37.608,157.132
C08503=1058.730,375.200,386.628,174.270,37.614,157.134
C08504=1058.738,375.447,386.589,174.275,37.621,157.135
C08505=1058.745,375.694,386.550,174.280,37.627,157.137
C08506=1058.752,375.940,386.510,174.286,37.633,157.138
C08507=1058.760,376.187,386.470,174.292,37.639,157.140
C08508=1058.767,376.433,386.430,174.297,37.645,157.142
C08509=1058.775,376.680,386.391,174.302,37.652,157.143
C08510=1058.782,376.927,386.351,174.307,37.658,157.145
C08511=1058.789,377.174,386.312,174.313,37.664,157.146
C08512=1058.797,377.421,386.272,174.318,37.670,157.148
C08513=1058.804,377.667,386.232,174.323,37.677,157.149
C08514=1058.812,377.914,386.192,174.328,37.683,157.151
C08515=1058.819,378.161,386.152,174.333,37.690,157.153
C08516=1058.827,378.407,386.113,174.339,37.696,157.154
C08517=1058.834,378.654,386.073,174.344,37.702,157.156
C08518=1058.841,378.900,386.033,174.350,37.709,157.157
C08519=1058.849,379.147,385.994,174.355,37.715,157.159
C08520=1058.857,379.393,385.953,174.360,37.722,157.161
C08521=1058.865,379.640,385.913,174.366,37.728,157.162
C08522=1058.872,379.887,385.873,174.371,37.734,157.164
C08523=1058.880,380.134,385.834,174.376,37.741,157.165
C08524=1058.887,380.380,385.794,174.381,37.747,157.167
C08525=1058.895,380.627,385.752,174.388,37.754,157.169
C08526=1058.902,380.873,385.713,174.393,37.760,157.170
C08527=1058.910,381.120,385.673,174.398,37.767,157.172
C08528=1058.917,381.367,385.632,174.403,37.773,157.174
C08529=1058.924,381.613,385.592,174.409,37.780,157.175
C08530=1058.932,381.860,385.552,174.414,37.786,157.177
C08531=1058.939,382.106,385.511,174.420,37.793,157.179
C08532=1058.947,382.353,385.471,174.426,37.800,157.180
C08533=1058.954,382.599,385.431,174.431,37.806,157.182
C08534=1058.961,382.846,385.390,174.436,37.813,157.184
C08535=1058.969,383.092,385.350,174.441,37.819,157.185
C08536=1058.977,383.339,385.309,174.448,37.826,157.187
C08537=1058.984,383.586,385.268,174.453,37.833,157.189
C08538=1058.992,383.831,385.228,174.458,37.839,157.190
C08539=1058.998,384.079,385.188,174.464,37.846,157.192
C08540=1059.007,384.325,385.147,174.470,37.853,157.194
C08541=1059.015,384.571,385.106,174.475,37.860,157.196
C08542=1059.022,384.818,385.065,174.481,37.866,157.197
C08543=1059.030,385.065,385.025,174.486,37.874,157.199
C08544=1059.037,385.311,384.984,174.492,37.880,157.201
C08545=1059.045,385.558,384.943,174.498,37.887,157.203
C08546=1059.053,385.804,384.903,174.503,37.894,157.204
C08547=1059.060,386.051,384.862,174.509,37.901,157.206
C08548=1059.068,386.296,384.821,174.515,37.908,157.208
C08549=1059.075,386.543,384.780,174.520,37.914,157.209
C08550=1059.083,386.789,384.739,174.527,37.921,157.211
C08551=1059.091,387.036,384.698,174.532,37.928,157.213
C08552=1059.100,387.341,384.648,174.539,37.937,157.215
C08553=1059.110,387.647,384.597,174.546,37.945,157.217
C08554=1059.119,387.951,384.546,174.553,37.954,157.220
C08555=1059.129,388.257,384.496,174.561,37.963,157.222
C08556=1059.137,388.503,384.454,174.566,37.970,157.224
C08557=1059.145,388.749,384.414,174.572,37.977,157.226
C08558=1059.152,388.996,384.372,174.578,37.984,157.227
C08559=1059.161,389.243,384.331,174.584,37.991,157.229
C08560=1059.168,389.490,384.290,174.590,37.998,157.231
C08561=1059.176,389.735,384.249,174.596,38.005,157.233
C08562=1059.184,389.982,384.208,174.601,38.012,157.235
C08563=1059.192,390.228,384.167,174.607,38.019,157.236
C08564=1059.199,390.474,384.125,174.613,38.026,157.238
C08565=1059.207,390.721,384.083,174.619,38.033,157.240
C08566=1059.215,390.967,384.041,174.625,38.040,157.242
C08567=1059.223,391.214,384.001,174.631,38.047,157.244
C08568=1059.230,391.460,383.959,174.637,38.055,157.246
C08569=1059.238,391.706,383.918,174.643,38.061,157.247
C08570=1059.247,391.953,383.876,174.649,38.069,157.249
C08571=1059.254,392.199,383.835,174.655,38.076,157.251
C08572=1059.262,392.445,383.793,174.661,38.084,157.253
C08573=1059.269,392.691,383.751,174.668,38.091,157.255
C08574=1059.278,392.938,383.710,174.673,38.098,157.257
C08575=1059.285,393.184,383.668,174.680,38.105,157.259
C08576=1059.293,393.430,383.626,174.685,38.113,157.261
C08577=1059.301,393.677,383.584,174.692,38.120,157.263
C08578=1059.308,393.923,383.542,174.697,38.127,157.265
C08579=1059.316,394.169,383.500,174.704,38.135,157.267
C08580=1059.324,394.416,383.458,174.709,38.142,157.268
C08581=1059.333,394.662,383.417,174.716,38.150,157.270
C08582=1059.340,394.908,383.375,174.722,38.157,157.272
C08583=1059.348,395.154,383.333,174.728,38.165,157.274
C08584=1059.356,395.400,383.291,174.735,38.172,157.276
C08585=1059.364,395.647,383.248,174.740,38.180,157.278
C08586=1059.372,395.893,383.206,174.747,38.187,157.280
C08587=1059.380,396.140,383.164,174.753,38.195,157.282
C08588=1059.388,396.386,383.122,174.759,38.202,157.284
C08589=1059.396,396.632,383.080,174.766,38.210,157.286
C08590=1059.403,396.878,383.038,174.772,38.218,157.288
C08591=1059.412,397.124,382.995,174.778,38.225,157.290
C08592=1059.419,397.370,382.953,174.784,38.233,157.292
C08593=1059.428,397.617,382.911,174.791,38.241,157.294
C08594=1059.435,397.863,382.869,174.797,38.248,157.296
C08595=1059.444,398.109,382.826,174.803,38.256,157.298
C08596=1059.451,398.355,382.784,174.810,38.264,157.300
C08597=1059.460,398.602,382.741,174.816,38.272,157.302
C08598=1059.468,398.848,382.698,174.822,38.280,157.304
C08599=1059.475,399.094,382.656,174.829,38.287,157.306
C08600=1059.483,399.340,382.613,174.835,38.295,157.309
C08601=1059.492,399.587,382.570,174.841,38.303,157.311
C08602=1059.499,399.832,382.528,174.848,38.311,157.313
C08603=1059.508,400.079,382.485,174.855,38.318,157.315
C08604=1059.516,400.325,382.442,174.861,38.326,157.317
C08605=1059.523,400.570,382.399,174.867,38.334,157.319
C08606=1059.532,400.817,382.357,174.874,38.342,157.321
C08607=1059.540,401.063,382.314,174.881,38.350,157.323
C08608=1059.551,401.386,382.258,174.889,38.361,157.326
C08609=1059.561,401.708,382.201,174.897,38.372,157.329
C08610=1059.572,402.031,382.145,174.907,38.382,157.331
C08611=1059.583,402.353,382.089,174.915,38.392,157.334
C08612=1059.591,402.600,382.046,174.922,38.401,157.337
C08613=1059.599,402.846,382.003,174.929,38.409,157.339
C08614=1059.608,403.092,381.960,174.936,38.417,157.341
C08615=1059.615,403.338,381.916,174.941,38.425,157.343
C08616=1059.624,403.584,381.873,174.948,38.433,157.345
C08617=1059.632,403.830,381.830,174.955,38.442,157.347
C08618=1059.640,404.077,381.787,174.962,38.450,157.350
C08619=1059.648,404.321,381.743,174.969,38.458,157.352
C08620=1059.656,404.568,381.700,174.976,38.466,157.354
C08621=1059.665,404.814,381.657,174.983,38.474,157.356
C08622=1059.672,405.060,381.613,174.990,38.483,157.358
C08623=1059.681,405.306,381.570,174.996,38.491,157.361
C08624=1059.689,405.552,381.526,175.002,38.500,157.363
C08625=1059.698,405.799,381.482,175.009,38.508,157.365
C08626=1059.706,406.045,381.439,175.016,38.516,157.367
C08627=1059.715,406.290,381.395,175.023,38.525,157.370
C08628=1059.722,406.537,381.351,175.030,38.534,157.372
C08629=1059.730,406.783,381.307,175.037,38.542,157.374
C08630=1059.739,407.029,381.264,175.044,38.550,157.377
C08631=1059.747,407.274,381.220,175.051,38.559,157.379
C08632=1059.755,407.521,381.176,175.058,38.567,157.381
C08633=1059.764,407.766,381.132,175.065,38.576,157.384
C08634=1059.771,408.012,381.089,175.072,38.585,157.386
C08635=1059.779,408.258,381.044,175.079,38.593,157.388
C08636=1059.789,408.504,381.000,175.086,38.602,157.391
C08637=1059.797,408.750,380.956,175.093,38.610,157.393
C08638=1059.805,408.996,380.912,175.100,38.619,157.395
C08639=1059.813,409.242,380.868,175.107,38.628,157.398
C08640=1059.822,409.488,380.824,175.116,38.637,157.400
C08641=1059.830,409.734,380.779,175.123,38.646,157.402
C08642=1059.839,409.980,380.736,175.130,38.655,157.405
C08643=1059.848,410.226,380.691,175.137,38.663,157.407
C08644=1059.855,410.472,380.647,175.144,38.672,157.410
C08645=1059.864,410.718,380.604,175.151,38.681,157.412
C08646=1059.873,410.964,380.558,175.158,38.690,157.414
C08647=1059.881,411.209,380.514,175.166,38.699,157.417
C08648=1059.890,411.456,380.469,175.174,38.708,157.419
C08649=1059.899,411.701,380.425,175.181,38.716,157.422
C08650=1059.907,411.947,380.381,175.188,38.725,157.424
C08651=1059.915,412.193,380.336,175.195,38.734,157.427
C08652=1059.924,412.439,380.293,175.203,38.743,157.429
C08653=1059.933,412.685,380.247,175.210,38.753,157.432
C08654=1059.941,412.930,380.203,175.218,38.762,157.434
C08655=1059.950,413.177,380.158,175.225,38.770,157.437
C08656=1059.959,413.423,380.113,175.233,38.780,157.439
C08657=1059.968,413.668,380.069,175.240,38.789,157.442
C08658=1059.976,413.915,380.024,175.248,38.798,157.444
C08659=1059.985,414.160,379.979,175.256,38.807,157.447
C08660=1059.994,414.406,379.935,175.263,38.816,157.449
C08661=1060.003,414.652,379.889,175.270,38.826,157.452
C08662=1060.011,414.897,379.844,175.279,38.835,157.454
C08663=1060.020,415.144,379.799,175.286,38.845,157.457
C08664=1060.031,415.471,379.739,175.296,38.857,157.460
C08665=1060.043,415.799,379.678,175.306,38.870,157.464
C08666=1060.054,416.127,379.618,175.317,38.882,157.467
C08667=1060.065,416.455,379.558,175.328,38.895,157.471
C08668=1060.074,416.700,379.513,175.335,38.904,157.473
C08669=1060.083,416.946,379.467,175.343,38.914,157.476
C08670=1060.092,417.192,379.422,175.351,38.923,157.479
C08671=1060.100,417.437,379.377,175.359,38.932,157.481
C08672=1060.109,417.683,379.331,175.367,38.942,157.484
C08673=1060.118,417.929,379.286,175.375,38.952,157.487
C08674=1060.127,418.175,379.240,175.383,38.962,157.490
C08675=1060.136,418.421,379.195,175.391,38.971,157.492
C08676=1060.145,418.666,379.150,175.398,38.981,157.495
C08677=1060.154,418.912,379.103,175.407,38.991,157.498
C08678=1060.162,419.157,379.058,175.415,39.000,157.500
C08679=1060.171,419.403,379.012,175.423,39.010,157.503
C08680=1060.180,419.649,378.967,175.432,39.020,157.506
C08681=1060.190,419.895,378.920,175.439,39.030,157.509
C08682=1060.199,420.140,378.875,175.448,39.040,157.511
C08683=1060.208,420.386,378.828,175.456,39.050,157.514
C08684=1060.216,420.632,378.783,175.464,39.060,157.517
C08685=1060.226,420.877,378.737,175.472,39.069,157.520
C08686=1060.234,421.123,378.691,175.481,39.080,157.523
C08687=1060.243,421.368,378.645,175.489,39.090,157.525
C08688=1060.252,421.614,378.598,175.497,39.100,157.528
C08689=1060.261,421.860,378.552,175.506,39.110,157.531
C08690=1060.270,422.105,378.506,175.515,39.120,157.534
C08691=1060.279,422.350,378.460,175.522,39.130,157.537
C08692=1060.288,422.596,378.413,175.531,39.140,157.540
C08693=1060.296,422.841,378.367,175.540,39.150,157.543
C08694=1060.306,423.086,378.321,175.548,39.161,157.546
C08695=1060.315,423.332,378.273,175.556,39.171,157.548
C08696=1060.324,423.578,378.227,175.565,39.181,157.551
C08697=1060.333,423.823,378.181,175.573,39.192,157.554
C08698=1060.342,424.068,378.134,175.582,39.202,157.557
C08699=1060.352,424.314,378.088,175.591,39.212,157.560
C08700=1060.360,424.560,378.041,175.600,39.222,157.563
C08701=1060.370,424.805,377.995,175.609,39.233,157.566
C08702=1060.379,425.050,377.948,175.617,39.243,157.569
C08703=1060.388,425.296,377.901,175.626,39.254,157.572
C08704=1060.397,425.541,377.854,175.634,39.265,157.575
C08705=1060.407,425.787,377.807,175.643,39.275,157.578
C08706=1060.416,426.032,377.760,175.652,39.286,157.581
C08707=1060.425,426.277,377.714,175.661,39.296,157.584
C08708=1060.434,426.523,377.667,175.670,39.307,157.587
C08709=1060.444,426.768,377.620,175.679,39.318,157.590
C08710=1060.453,427.014,377.573,175.688,39.329,157.594
C08711=1060.462,427.259,377.525,175.698,39.339,157.597
C08712=1060.472,427.505,377.479,175.707,39.350,157.600
C08713=1060.481,427.749,377.431,175.715,39.361,157.603
C08714=1060.490,427.995,377.383,175.724,39.372,157.606
C08715=1060.499,428.240,377.336,175.734,39.383,157.609
C08716=1060.509,428.485,377.289,175.743,39.394,157.612
C08717=1060.518,428.730,377.241,175.752,39.404,157.615
C08718=1060.528,428.976,377.193,175.761,39.415,157.619
C08719=1060.538,429.221,377.146,175.771,39.427,157.622
C08720=1060.551,429.570,377.079,175.783,39.442,157.626
C08721=1060.564,429.919,377.011,175.797,39.458,157.631
C08722=1060.577,430.267,376.943,175.810,39.474,157.636
C08723=1060.591,430.616,376.875,175.824,39.490,157.640
C08724=1060.601,430.861,376.828,175.833,39.501,157.644
C08725=1060.610,431.106,376.779,175.843,39.512,157.647
C08726=1060.619,431.351,376.732,175.852,39.524,157.650
C08727=1060.629,431.597,376.684,175.861,39.535,157.654
C08728=1060.638,431.842,376.635,175.872,39.546,157.657
C08729=1060.648,432.087,376.587,175.881,39.558,157.660
C08730=1060.658,432.332,376.539,175.890,39.570,157.664
C08731=1060.667,432.577,376.491,175.901,39.581,157.667
C08732=1060.676,432.822,376.443,175.910,39.592,157.670
C08733=1060.686,433.067,376.394,175.920,39.604,157.674
C08734=1060.696,433.312,376.346,175.930,39.616,157.677
C08735=1060.706,433.557,376.297,175.940,39.627,157.681
C08736=1060.715,433.802,376.249,175.949,39.639,157.684
C08737=1060.725,434.047,376.200,175.960,39.651,157.688
C08738=1060.735,434.292,376.152,175.969,39.662,157.691
C08739=1060.745,434.537,376.103,175.980,39.674,157.695
C08740=1060.754,434.782,376.055,175.989,39.686,157.698
C08741=1060.764,435.027,376.006,176.000,39.698,157.702
C08742=1060.775,435.273,375.957,176.009,39.710,157.705
C08743=1060.784,435.518,375.909,176.020,39.722,157.709
C08744=1060.793,435.763,375.860,176.030,39.733,157.712
C08745=1060.803,436.007,375.810,176.040,39.745,157.716
C08746=1060.813,436.252,375.762,176.050,39.758,157.719
C08747=1060.823,436.497,375.713,176.061,39.770,157.723
C08748=1060.834,436.742,375.664,176.071,39.782,157.727
C08749=1060.843,436.987,375.615,176.081,39.794,157.730
C08750=1060.853,437.231,375.566,176.092,39.806,157.734
C08751=1060.864,437.477,375.517,176.103,39.818,157.738
C08752=1060.874,437.721,375.468,176.113,39.830,157.741
C08753=1060.883,437.966,375.418,176.123,39.843,157.745
C08754=1060.893,438.212,375.369,176.134,39.855,157.749
C08755=1060.904,438.456,375.320,176.145,39.868,157.752
C08756=1060.914,438.701,375.270,176.156,39.880,157.756
C08757=1060.924,438.946,375.221,176.166,39.893,157.760
C08758=1060.934,439.190,375.171,176.177,39.905,157.764
C08759=1060.944,439.435,375.122,176.188,39.918,157.768
C08760=1060.954,439.680,375.072,176.199,39.930,157.771
C08761=1060.964,439.925,375.022,176.210,39.943,157.775
C08762=1060.974,440.170,374.972,176.221,39.956,157.779
C08763=1060.984,440.415,374.923,176.232,39.968,157.783
C08764=1060.995,440.659,374.872,176.243,39.981,157.787
C08765=1061.005,440.904,374.823,176.254,39.993,157.791
C08766=1061.015,441.149,374.773,176.265,40.006,157.795
C08767=1061.025,441.393,374.722,176.276,40.019,157.798
C08768=1061.036,441.638,374.673,176.287,40.032,157.802
C08769=1061.046,441.883,374.622,176.298,40.045,157.806
C08770=1061.056,442.128,374.572,176.309,40.058,157.810
C08771=1061.066,442.372,374.522,176.321,40.071,157.814
C08772=1061.077,442.617,374.472,176.332,40.085,157.818
C08773=1061.087,442.862,374.421,176.343,40.098,157.822
C08774=1061.098,443.106,374.371,176.354,40.110,157.826
C08775=1061.108,443.351,374.320,176.367,40.124,157.831
C08776=1061.117,443.562,374.277,176.376,40.135,157.834
C08777=1061.126,443.773,374.233,176.386,40.147,157.838
C08778=1061.135,443.983,374.189,176.397,40.158,157.841
C08779=1061.144,444.195,374.146,176.407,40.170,157.845
C08780=1061.153,444.406,374.101,176.416,40.181,157.848
C08781=1061.162,444.616,374.058,176.427,40.193,157.852
C08782=1061.171,444.828,374.014,176.437,40.205,157.855
C08783=1061.180,445.039,373.970,176.447,40.216,157.859
C08784=1061.191,445.283,373.920,176.459,40.230,157.863
C08785=1061.202,445.528,373.868,176.470,40.244,157.868
C08786=1061.212,445.772,373.817,176.483,40.257,157.872
C08787=1061.223,446.016,373.766,176.495,40.271,157.876
C08788=1061.233,446.261,373.715,176.507,40.284,157.880
C08789=1061.245,446.505,373.664,176.519,40.298,157.885
C08790=1061.255,446.750,373.613,176.531,40.312,157.889
C08791=1061.266,446.994,373.561,176.544,40.326,157.893
C08792=1061.277,447.237,373.511,176.556,40.340,157.898
C08793=1061.287,447.480,373.460,176.568,40.353,157.902
C08794=1061.301,447.724,373.410,176.580,40.367,157.906
C08795=1061.313,447.969,373.360,176.593,40.380,157.910
C08796=1061.328,448.213,373.311,176.605,40.393,157.915
C08797=1061.342,448.457,373.263,176.619,40.406,157.919
C08798=1061.358,448.701,373.215,176.631,40.418,157.923
C08799=1061.375,448.946,373.168,176.644,40.430,157.927
C08800=1061.393,449.191,373.121,176.656,40.443,157.931
C08801=1061.412,449.437,373.075,176.669,40.454,157.934
C08802=1061.430,449.682,373.030,176.682,40.466,157.938
C08803=1061.451,449.927,372.985,176.695,40.477,157.942
C08804=1061.119,449.938,372.710,176.690,40.593,157.974
C08805=1061.098,449.692,372.754,176.677,40.582,157.970
C08806=1061.078,449.447,372.800,176.664,40.570,157.966
C08807=1061.059,449.202,372.845,176.651,40.559,157.962
C08808=1061.042,448.957,372.891,176.637,40.547,157.958
C08809=1061.025,448.712,372.939,176.624,40.534,157.954
C08810=1061.009,448.467,372.987,176.612,40.522,157.950
C08811=1060.994,448.222,373.035,176.598,40.509,157.946
C08812=1060.979,447.979,373.084,176.586,40.497,157.942
C08813=1060.966,447.735,373.134,176.573,40.483,157.938
C08814=1060.954,447.491,373.183,176.561,40.470,157.934
C08815=1060.942,447.247,373.234,176.548,40.457,157.929
C08816=1060.931,447.005,373.285,176.537,40.443,157.925
C08817=1060.921,446.760,373.337,176.524,40.429,157.921
C08818=1060.910,446.515,373.388,176.511,40.415,157.916
C08819=1060.899,446.271,373.439,176.500,40.401,157.912
C08820=1060.888,446.026,373.490,176.487,40.388,157.908
C08821=1060.878,445.782,373.542,176.476,40.374,157.903
C08822=1060.867,445.538,373.592,176.463,40.361,157.899
C08823=1060.856,445.294,373.644,176.452,40.347,157.895
C08824=1060.845,445.049,373.694,176.439,40.333,157.891
C08825=1060.828,444.646,373.779,176.420,40.311,157.884
C08826=1060.811,444.243,373.862,176.400,40.289,157.877
C08827=1060.793,443.841,373.946,176.380,40.267,157.870
C08828=1060.776,443.438,374.029,176.361,40.245,157.863
C08829=1060.765,443.194,374.080,176.350,40.232,157.859
C08830=1060.755,442.949,374.130,176.339,40.219,157.855
C08831=1060.744,442.705,374.181,176.326,40.206,157.851
C08832=1060.734,442.459,374.231,176.315,40.193,157.847
C08833=1060.723,442.215,374.281,176.304,40.180,157.843
C08834=1060.713,441.971,374.332,176.293,40.167,157.839
C08835=1060.703,441.726,374.381,176.282,40.154,157.835
C08836=1060.693,441.481,374.432,176.270,40.141,157.831
C08837=1060.683,441.237,374.482,176.258,40.128,157.827
C08838=1060.672,440.992,374.533,176.247,40.115,157.823
C08839=1060.662,440.747,374.582,176.236,40.103,157.819
C08840=1060.652,440.502,374.632,176.225,40.090,157.815
C08841=1060.641,440.258,374.682,176.214,40.077,157.812
C08842=1060.631,440.013,374.732,176.203,40.065,157.808
C08843=1060.621,439.768,374.782,176.192,40.052,157.804
C08844=1060.611,439.523,374.831,176.181,40.040,157.800
C08845=1060.601,439.279,374.881,176.170,40.027,157.796
C08846=1060.591,439.033,374.931,176.160,40.015,157.792
C08847=1060.581,438.789,374.980,176.149,40.002,157.789
C08848=1060.570,438.544,375.030,176.138,39.990,157.785
C08849=1060.561,438.299,375.079,176.127,39.978,157.781
C08850=1060.551,438.055,375.129,176.116,39.965,157.777
C08851=1060.540,437.810,375.178,176.105,39.953,157.774
C08852=1060.531,437.565,375.227,176.096,39.940,157.770
C08853=1060.520,437.319,375.277,176.085,39.928,157.766
C08854=1060.510,437.075,375.326,176.074,39.916,157.763
C08855=1060.500,436.830,375.375,176.063,39.904,157.759
C08856=1060.490,436.585,375.424,176.054,39.892,157.755
C08857=1060.480,436.340,375.473,176.043,39.880,157.752
C08858=1060.470,436.096,375.522,176.032,39.868,157.748
C08859=1060.460,435.851,375.571,176.022,39.856,157.745
C08860=1060.450,435.605,375.620,176.012,39.844,157.741
C08861=1060.440,435.360,375.668,176.002,39.833,157.737
C08862=1060.430,435.116,375.717,175.991,39.820,157.734
C08863=1060.420,434.871,375.766,175.982,39.809,157.730
C08864=1060.410,434.626,375.814,175.971,39.797,157.727
C08865=1060.401,434.381,375.863,175.961,39.785,157.723
C08866=1060.391,434.136,375.912,175.951,39.774,157.720
C08867=1060.381,433.891,375.960,175.940,39.762,157.716
C08868=1060.371,433.646,376.009,175.931,39.750,157.713
C08869=1060.362,433.401,376.057,175.920,39.738,157.709
C08870=1060.352,433.156,376.106,175.911,39.727,157.706
C08871=1060.343,432.911,376.155,175.901,39.715,157.703
C08872=1060.333,432.665,376.203,175.891,39.704,157.699
C08873=1060.324,432.420,376.251,175.882,39.692,157.696
C08874=1060.314,432.175,376.300,175.872,39.681,157.692
C08875=1060.304,431.930,376.347,175.862,39.669,157.689
C08876=1060.295,431.685,376.396,175.852,39.658,157.686
C08877=1060.284,431.439,376.443,175.843,39.646,157.682
C08878=1060.275,431.195,376.491,175.833,39.635,157.679
C08879=1060.266,430.950,376.539,175.823,39.624,157.676
C08880=1060.256,430.705,376.588,175.814,39.613,157.672
C08881=1060.243,430.353,376.656,175.800,39.597,157.668
C08882=1060.229,430.003,376.725,175.787,39.581,157.663
C08883=1060.216,429.653,376.792,175.773,39.565,157.658
C08884=1060.202,429.302,376.861,175.760,39.549,157.654
C08885=1060.192,429.056,376.908,175.750,39.538,157.650
C08886=1060.183,428.812,376.956,175.741,39.528,157.647
C08887=1060.174,428.566,377.004,175.732,39.516,157.644
C08888=1060.164,428.321,377.051,175.723,39.506,157.641
C08889=1060.155,428.076,377.098,175.713,39.494,157.638
C08890=1060.146,427.830,377.145,175.704,39.484,157.635
C08891=1060.136,427.585,377.192,175.695,39.473,157.631
C08892=1060.127,427.339,377.240,175.686,39.462,157.628
C08893=1060.118,427.094,377.288,175.677,39.451,157.625
C08894=1060.108,426.849,377.334,175.668,39.441,157.622
C08895=1060.099,426.604,377.382,175.659,39.430,157.619
C08896=1060.090,426.358,377.429,175.650,39.419,157.616
C08897=1060.080,426.113,377.475,175.641,39.409,157.613
C08898=1060.071,425.867,377.523,175.632,39.398,157.610
C08899=1060.062,425.622,377.569,175.623,39.387,157.607
C08900=1060.053,425.377,377.616,175.614,39.377,157.604
C08901=1060.043,425.131,377.663,175.605,39.367,157.601
C08902=1060.034,424.886,377.710,175.596,39.356,157.598
C08903=1060.024,424.640,377.757,175.588,39.346,157.595
C08904=1060.016,424.395,377.804,175.579,39.336,157.592
C08905=1060.006,424.150,377.850,175.570,39.325,157.589
C08906=1059.996,423.904,377.897,175.561,39.315,157.586
C08907=1059.988,423.658,377.943,175.553,39.304,157.583
C08908=1059.979,423.413,377.990,175.544,39.294,157.580
C08909=1059.970,423.168,378.036,175.536,39.284,157.577
C08910=1059.961,422.922,378.082,175.527,39.274,157.574
C08911=1059.952,422.676,378.130,175.518,39.264,157.571
C08912=1059.942,422.431,378.176,175.509,39.253,157.568
C08913=1059.933,422.186,378.222,175.502,39.244,157.566
C08914=1059.924,421.940,378.269,175.493,39.233,157.563
C08915=1059.915,421.694,378.314,175.484,39.223,157.560
C08916=1059.907,421.449,378.361,175.476,39.213,157.557
C08917=1059.898,421.204,378.407,175.468,39.203,157.554
C08918=1059.888,420.959,378.453,175.459,39.193,157.551
C08919=1059.880,420.712,378.499,175.451,39.183,157.548
C08920=1059.871,420.467,378.545,175.443,39.173,157.546
C08921=1059.863,420.221,378.591,175.434,39.163,157.543
C08922=1059.853,419.975,378.638,175.426,39.153,157.540
C08923=1059.844,419.729,378.683,175.418,39.143,157.537
C08924=1059.834,419.484,378.729,175.410,39.134,157.534
C08925=1059.825,419.238,378.775,175.401,39.124,157.532
C08926=1059.817,418.992,378.820,175.394,39.115,157.529
C08927=1059.807,418.747,378.866,175.385,39.105,157.526
C08928=1059.800,418.502,378.912,175.377,39.095,157.523
C08929=1059.791,418.256,378.957,175.369,39.086,157.521
C08930=1059.782,418.010,379.003,175.361,39.076,157.518
C08931=1059.773,417.764,379.048,175.353,39.066,157.515
C08932=1059.764,417.519,379.093,175.345,39.056,157.513
C08933=1059.754,417.273,379.140,175.337,39.047,157.510
C08934=1059.745,417.028,379.185,175.330,39.038,157.507
C08935=1059.737,416.782,379.230,175.321,39.028,157.505
C08936=1059.728,416.536,379.275,175.314,39.019,157.502
C08937=1059.717,416.207,379.336,175.302,39.006,157.499
C08938=1059.705,415.877,379.397,175.292,38.993,157.495
C08939=1059.693,415.547,379.458,175.282,38.981,157.491
C08940=1059.682,415.217,379.518,175.272,38.968,157.488
C08941=1059.673,414.971,379.564,175.263,38.959,157.485
C08942=1059.665,414.725,379.608,175.256,38.949,157.483
C08943=1059.656,414.480,379.654,175.248,38.941,157.480
C08944=1059.647,414.234,379.699,175.240,38.931,157.478
C08945=1059.639,413.988,379.743,175.233,38.922,157.475
C08946=1059.630,413.742,379.789,175.225,38.913,157.473
C08947=1059.622,413.496,379.833,175.217,38.903,157.470
C08948=1059.612,413.250,379.877,175.210,38.895,157.468
C08949=1059.603,413.004,379.923,175.203,38.886,157.465
C08950=1059.595,412.759,379.967,175.195,38.876,157.463
C08951=1059.587,412.512,380.012,175.187,38.867,157.460
C08952=1059.577,412.268,380.056,175.180,38.859,157.458
C08953=1059.569,412.021,380.101,175.172,38.850,157.455
C08954=1059.561,411.775,380.145,175.165,38.841,157.453
C08955=1059.551,411.529,380.189,175.158,38.832,157.450
C08956=1059.543,411.283,380.234,175.150,38.823,157.448
C08957=1059.534,411.038,380.279,175.143,38.814,157.445
C08958=1059.526,410.792,380.323,175.135,38.805,157.443
C08959=1059.517,410.546,380.367,175.128,38.796,157.441
C08960=1059.509,410.300,380.412,175.121,38.787,157.438
C08961=1059.501,410.054,380.456,175.114,38.778,157.436
C08962=1059.492,409.809,380.500,175.106,38.770,157.433
C08963=1059.483,409.562,380.544,175.099,38.761,157.431
C08964=1059.475,409.316,380.588,175.092,38.752,157.429
C08965=1059.467,409.071,380.632,175.084,38.744,157.426
C08966=1059.458,408.824,380.677,175.077,38.735,157.424
C08967=1059.450,408.578,380.721,175.070,38.726,157.421
C08968=1059.441,408.333,380.765,175.063,38.718,157.419
C08969=1059.433,408.087,380.808,175.056,38.709,157.417
C08970=1059.425,407.840,380.853,175.049,38.701,157.414
C08971=1059.416,407.595,380.897,175.042,38.692,157.412
C08972=1059.408,407.348,380.940,175.035,38.683,157.410
C08973=1059.400,407.103,380.985,175.028,38.675,157.407
C08974=1059.391,406.857,381.028,175.021,38.666,157.405
C08975=1059.383,406.611,381.072,175.014,38.658,157.403
C08976=1059.376,406.364,381.116,175.007,38.650,157.401
C08977=1059.367,406.119,381.159,175.000,38.641,157.398
C08978=1059.359,405.873,381.203,174.993,38.633,157.396
C08979=1059.350,405.627,381.247,174.986,38.624,157.394
C08980=1059.342,405.380,381.291,174.979,38.616,157.391
C08981=1059.333,405.134,381.334,174.972,38.607,157.389
C08982=1059.326,404.888,381.377,174.966,38.599,157.387
C08983=1059.317,404.642,381.421,174.959,38.591,157.385
C08984=1059.309,404.396,381.465,174.952,38.583,157.383
C08985=1059.301,404.150,381.508,174.945,38.575,157.380
C08986=1059.293,403.903,381.551,174.938,38.566,157.378
C08987=1059.284,403.657,381.595,174.931,38.558,157.376
C08988=1059.276,403.412,381.637,174.924,38.550,157.374
C08989=1059.269,403.166,381.681,174.917,38.542,157.372
C08990=1059.260,402.920,381.724,174.911,38.533,157.369
C08991=1059.252,402.674,381.767,174.904,38.525,157.367
C08992=1059.244,402.427,381.810,174.898,38.518,157.365
C08993=1059.233,402.103,381.868,174.889,38.507,157.362
C08994=1059.222,401.779,381.924,174.880,38.496,157.359
C08995=1059.211,401.455,381.980,174.871,38.486,157.357
C08996=1059.200,401.131,382.037,174.863,38.475,157.354
C08997=1059.192,400.884,382.079,174.856,38.467,157.352
C08998=1059.184,400.638,382.123,174.849,38.459,157.349
C08999=1059.176,400.392,382.166,174.843,38.451,157.347
C09000=1059.168,400.146,382.208,174.837,38.444,157.345
C09001=1059.160,399.900,382.251,174.830,38.436,157.343
C09002=1059.152,399.653,382.293,174.823,38.428,157.341
C09003=1059.143,399.407,382.336,174.816,38.420,157.339
C09004=1059.135,399.162,382.379,174.811,38.412,157.337
C09005=1059.128,398.915,382.422,174.804,38.404,157.335
C09006=1059.120,398.668,382.464,174.797,38.397,157.333
C09007=1059.112,398.422,382.507,174.791,38.389,157.331
C09008=1059.103,398.176,382.549,174.785,38.381,157.329
C09009=1059.096,397.930,382.592,174.778,38.374,157.327
C09010=1059.087,397.684,382.634,174.772,38.366,157.325
C09011=1059.079,397.437,382.677,174.766,38.358,157.323
C09012=1059.071,397.192,382.719,174.759,38.350,157.321
C09013=1059.063,396.945,382.762,174.753,38.343,157.319
C09014=1059.055,396.699,382.803,174.747,38.335,157.317
C09015=1059.047,396.452,382.846,174.740,38.328,157.315
C09016=1059.040,396.206,382.888,174.734,38.320,157.313
C09017=1059.031,395.960,382.930,174.728,38.313,157.311
C09018=1059.024,395.714,382.973,174.722,38.305,157.309
C09019=1059.015,395.468,383.015,174.715,38.297,157.307
C09020=1059.008,395.222,383.057,174.709,38.290,157.305
C09021=1059.000,394.975,383.099,174.703,38.282,157.303
C09022=1058.992,394.729,383.141,174.696,38.275,157.301
C09023=1058.984,394.483,383.183,174.691,38.267,157.299
C09024=1058.975,394.237,383.225,174.684,38.261,157.297
C09025=1058.968,393.990,383.266,174.679,38.253,157.295
C09026=1058.961,393.744,383.308,174.672,38.246,157.293
C09027=1058.952,393.498,383.350,174.665,38.238,157.291
C09028=1058.945,393.252,383.392,174.660,38.231,157.289
C09029=1058.937,393.006,383.434,174.653,38.224,157.287
C09030=1058.929,392.758,383.476,174.648,38.216,157.285
C09031=1058.921,392.513,383.517,174.641,38.209,157.284
C09032=1058.913,392.267,383.559,174.635,38.202,157.282
C09033=1058.905,392.019,383.601,174.629,38.195,157.280
C09034=1058.898,391.773,383.643,174.623,38.187,157.278
C09035=1058.890,391.528,383.684,174.617,38.180,157.276
C09036=1058.882,391.281,383.725,174.611,38.173,157.274
C09037=1058.874,391.034,383.768,174.605,38.166,157.272
C09038=1058.866,390.788,383.808,174.599,38.158,157.270
C09039=1058.858,390.542,383.850,174.594,38.151,157.268
C09040=1058.851,390.296,383.891,174.587,38.144,157.267
C09041=1058.843,390.050,383.933,174.582,38.137,157.265
C09042=1058.835,389.803,383.974,174.575,38.130,157.263
C09043=1058.828,389.556,384.016,174.570,38.123,157.261
C09044=1058.820,389.310,384.056,174.563,38.116,157.259
C09045=1058.811,389.064,384.098,174.558,38.109,157.257
C09046=1058.804,388.818,384.139,174.552,38.102,157.256
C09047=1058.796,388.571,384.179,174.546,38.095,157.254
C09048=1058.788,388.324,384.221,174.540,38.088,157.252
C09049=1058.778,388.017,384.272,174.533,38.079,157.250
C09050=1058.768,387.710,384.323,174.526,38.071,157.248
C09051=1058.759,387.403,384.374,174.518,38.062,157.245
C09052=1058.750,387.096,384.426,174.511,38.054,157.243
C09053=1058.742,386.850,384.466,174.506,38.047,157.241
C09054=1058.734,386.604,384.507,174.499,38.040,157.240
C09055=1058.726,386.357,384.548,174.494,38.033,157.238
C09056=1058.718,386.111,384.589,174.489,38.026,157.236
C09057=1058.711,385.864,384.630,174.482,38.019,157.234
C09058=1058.703,385.617,384.670,174.477,38.013,157.233
C09059=1058.695,385.371,384.711,174.471,38.006,157.231
C09060=1058.688,385.124,384.752,174.465,37.999,157.229
C09061=1058.680,384.878,384.793,174.460,37.992,157.227
C09062=1058.673,384.632,384.834,174.454,37.986,157.226
C09063=1058.665,384.385,384.874,174.449,37.979,157.224
C09064=1058.657,384.139,384.914,174.443,37.972,157.222
C09065=1058.650,383.892,384.955,174.437,37.965,157.221
C09066=1058.642,383.646,384.996,174.432,37.959,157.219
C09067=1058.635,383.399,385.036,174.427,37.952,157.217
C09068=1058.627,383.153,385.077,174.420,37.945,157.215
C09069=1058.619,382.906,385.117,174.415,37.939,157.214
C09070=1058.612,382.659,385.158,174.409,37.932,157.212
C09071=1058.605,382.414,385.198,174.404,37.926,157.210
C09072=1058.597,382.167,385.238,174.399,37.919,157.209
C09073=1058.590,381.920,385.280,174.392,37.912,157.207
C09074=1058.582,381.673,385.319,174.387,37.906,157.205
C09075=1058.575,381.428,385.360,174.382,37.899,157.204
C09076=1058.568,381.180,385.400,174.377,37.893,157.202
C09077=1058.560,380.933,385.440,174.371,37.886,157.200
C09078=1058.552,380.687,385.481,174.366,37.880,157.199
C09079=1058.545,380.441,385.521,174.360,37.873,157.197
C09080=1058.538,380.194,385.561,174.354,37.867,157.195
C09081=1058.530,379.947,385.601,174.349,37.860,157.194
C09082=1058.522,379.701,385.641,174.344,37.854,157.192
C09083=1058.515,379.454,385.681,174.339,37.848,157.191
C09084=1058.507,379.207,385.721,174.333,37.841,157.189
C09085=1058.499,378.961,385.761,174.327,37.835,157.187
C09086=1058.492,378.714,385.800,174.322,37.829,157.186
C09087=1058.485,378.467,385.840,174.317,37.822,157.184
C09088=1058.477,378.221,385.880,174.311,37.816,157.183
C09089=1058.470,377.974,385.920,174.306,37.810,157.181
C09090=1058.462,377.727,385.960,174.301,37.803,157.179
C09091=1058.454,377.481,386.000,174.296,37.797,157.178
C09092=1058.447,377.234,386.039,174.291,37.791,157.176
C09093=1058.439,376.987,386.079,174.285,37.785,157.175
C09094=1058.432,376.741,386.119,174.280,37.778,157.173
C09095=1058.425,376.494,386.159,174.274,37.772,157.172
C09096=1058.417,376.248,386.198,174.269,37.766,157.170
C09097=1058.410,376.001,386.238,174.264,37.760,157.168
C09098=1058.402,375.754,386.277,174.258,37.753,157.167
C09099=1058.395,375.508,386.317,174.253,37.747,157.165
C09100=1058.388,375.261,386.356,174.248,37.741,157.164
C09101=1058.380,375.014,386.396,174.243,37.735,157.162
C09102=1058.374,374.768,386.435,174.238,37.729,157.161
C09103=1058.366,374.521,386.475,174.232,37.723,157.159
C09104=1058.359,374.274,386.515,174.227,37.717,157.158
C09105=1058.350,373.998,386.559,174.222,37.709,157.156
C09106=1058.342,373.723,386.603,174.216,37.703,157.154
